Fanuc TP program (LS listing): hs0301h80.ls

/PROG  hs0301h80
/ATTR
COMMENT	= "19-03-01 10:31:46";
PROG_SIZE	= 0;
DEFAULT_GROUP	= 1, 1, *, *, *;
/APPL
    ARC Welding Equipment: 1, *, *, *, *;
/MN
   1:  CALL HOME_ALL;
   1:  UFRAME_NUM = 1;
   1:  UTOOL_NUM = 3;
   1:  COL GUARD ADJUST 150;
   1:  PR[91] = PR[90];
   1:  PR[GP1:91,1] = PR[GP1:90,1] + -1.621;
   1:  PR[GP1:91,2] = PR[GP1:90,2] + 0.568;
   1:  PR[GP1:91,3] = PR[GP1:90,3] + 0.915;
   1:  PR[92] = PR[91];
   1:  PR[GP1:92,3] = PR[GP1:92,3] + 50;
   1:J PR[92] 10% FINE;
   1:L PR[91] R[100]mm/sec CNT100;
   1:  CALL LASER_DRAHT_START;
   1:  PR[GP1:91,1] = PR[GP1:90,1] + -2.739;
   1:  PR[GP1:91,2] = PR[GP1:90,2] + 0.824;
   1:L PR[91] R[100]mm/sec CNT100;
   1:  PR[GP1:91,1] = PR[GP1:90,1] + -3.104;
   1:  PR[GP1:91,2] = PR[GP1:90,2] + 1.033;
   1:L PR[91] R[100]mm/sec CNT100;
   1:  PR[GP1:91,1] = PR[GP1:90,1] + -3.825;
   1:  PR[GP1:91,2] = PR[GP1:90,2] + 1.631;
   1:L PR[91] R[100]mm/sec CNT100;
   1:  PR[GP1:91,1] = PR[GP1:90,1] + -4.095;
   1:  PR[GP1:91,2] = PR[GP1:90,2] + 1.948;
   1:L PR[91] R[100]mm/sec CNT100;
   1:  PR[GP1:91,1] = PR[GP1:90,1] + -4.477;
   1:  PR[GP1:91,2] = PR[GP1:90,2] + 2.812;
   1:L PR[91] R[100]mm/sec CNT100;
   1:  PR[GP1:91,1] = PR[GP1:90,1] + -6.542;
   1:  PR[GP1:91,2] = PR[GP1:90,2] + 8.483;
   1:L PR[91] R[100]mm/sec CNT100;
   1:  PR[GP1:91,1] = PR[GP1:90,1] + -6.656;
   1:  PR[GP1:91,2] = PR[GP1:90,2] + 8.860;
   1:L PR[91] R[100]mm/sec CNT100;
   1:  PR[GP1:91,1] = PR[GP1:90,1] + -6.677;
   1:  PR[GP1:91,2] = PR[GP1:90,2] + 8.904;
   1:L PR[91] R[100]mm/sec CNT100;
   1:  PR[GP1:91,1] = PR[GP1:90,1] + -10.354;
   1:  PR[GP1:91,2] = PR[GP1:90,2] + 13.473;
   1:L PR[91] R[100]mm/sec CNT100;
   1:  PR[GP1:91,1] = PR[GP1:90,1] + -10.502;
   1:  PR[GP1:91,2] = PR[GP1:90,2] + 13.689;
   1:L PR[91] R[100]mm/sec CNT100;
   1:  PR[GP1:91,1] = PR[GP1:90,1] + -10.528;
   1:  PR[GP1:91,2] = PR[GP1:90,2] + 13.715;
   1:L PR[91] R[100]mm/sec CNT100;
   1:  PR[GP1:91,1] = PR[GP1:90,1] + -15.483;
   1:  PR[GP1:91,2] = PR[GP1:90,2] + 16.854;
   1:L PR[91] R[100]mm/sec CNT100;
   1:  PR[GP1:91,1] = PR[GP1:90,1] + -15.694;
   1:  PR[GP1:91,2] = PR[GP1:90,2] + 17.011;
   1:L PR[91] R[100]mm/sec CNT100;
   1:  PR[GP1:91,1] = PR[GP1:90,1] + -15.726;
   1:  PR[GP1:91,2] = PR[GP1:90,2] + 17.028;
   1:L PR[91] R[100]mm/sec CNT100;
   1:  PR[GP1:91,1] = PR[GP1:90,1] + -21.429;
   1:  PR[GP1:91,2] = PR[GP1:90,2] + 18.400;
   1:L PR[91] R[100]mm/sec CNT100;
   1:  PR[GP1:91,1] = PR[GP1:90,1] + -21.680;
   1:  PR[GP1:91,2] = PR[GP1:90,2] + 18.481;
   1:L PR[91] R[100]mm/sec CNT100;
   1:  PR[GP1:91,1] = PR[GP1:90,1] + -21.714;
   1:  PR[GP1:91,2] = PR[GP1:90,2] + 18.486;
   1:L PR[91] R[100]mm/sec CNT100;
   1:  PR[GP1:91,1] = PR[GP1:90,1] + -27.555;
   1:  PR[GP1:91,2] = PR[GP1:90,2] + 17.945;
   1:L PR[91] R[100]mm/sec CNT100;
   1:  PR[GP1:91,1] = PR[GP1:90,1] + -27.820;
   1:  PR[GP1:91,2] = PR[GP1:90,2] + 17.941;
   1:L PR[91] R[100]mm/sec CNT100;
   1:  PR[GP1:91,1] = PR[GP1:90,1] + -27.854;
   1:  PR[GP1:91,2] = PR[GP1:90,2] + 17.935;
   1:L PR[91] R[100]mm/sec CNT100;
   1:  PR[GP1:91,1] = PR[GP1:90,1] + -33.208;
   1:  PR[GP1:91,2] = PR[GP1:90,2] + 15.538;
   1:L PR[91] R[100]mm/sec CNT100;
   1:  PR[GP1:91,1] = PR[GP1:90,1] + -33.458;
   1:  PR[GP1:91,2] = PR[GP1:90,2] + 15.449;
   1:L PR[91] R[100]mm/sec CNT100;
   1:  PR[GP1:91,1] = PR[GP1:90,1] + -33.487;
   1:  PR[GP1:91,2] = PR[GP1:90,2] + 15.433;
   1:L PR[91] R[100]mm/sec CNT100;
   1:  PR[GP1:91,1] = PR[GP1:90,1] + -37.782;
   1:  PR[GP1:91,2] = PR[GP1:90,2] + 11.437;
   1:L PR[91] R[100]mm/sec CNT100;
   1:  PR[GP1:91,1] = PR[GP1:90,1] + -37.990;
   1:  PR[GP1:91,2] = PR[GP1:90,2] + 11.272;
   1:L PR[91] R[100]mm/sec CNT100;
   1:  PR[GP1:91,1] = PR[GP1:90,1] + -38.012;
   1:  PR[GP1:91,2] = PR[GP1:90,2] + 11.247;
   1:L PR[91] R[100]mm/sec CNT100;
   1:  PR[GP1:91,1] = PR[GP1:90,1] + -40.788;
   1:  PR[GP1:91,2] = PR[GP1:90,2] + 6.079;
   1:L PR[91] R[100]mm/sec CNT100;
   1:  PR[GP1:91,1] = PR[GP1:90,1] + -40.932;
   1:  PR[GP1:91,2] = PR[GP1:90,2] + 5.855;
   1:L PR[91] R[100]mm/sec CNT100;
   1:  PR[GP1:91,1] = PR[GP1:90,1] + -40.945;
   1:  PR[GP1:91,2] = PR[GP1:90,2] + 5.826;
   1:L PR[91] R[100]mm/sec CNT100;
   1:  PR[GP1:91,1] = PR[GP1:90,1] + -41.904;
   1:  PR[GP1:91,2] = PR[GP1:90,2] + 0.038;
   1:L PR[91] R[100]mm/sec CNT100;
   1:  PR[GP1:91,1] = PR[GP1:90,1] + -41.969;
   1:  PR[GP1:91,2] = PR[GP1:90,2] + -0.221;
   1:L PR[91] R[100]mm/sec CNT100;
   1:  PR[GP1:91,1] = PR[GP1:90,1] + -41.972;
   1:  PR[GP1:91,2] = PR[GP1:90,2] + -0.252;
   1:L PR[91] R[100]mm/sec CNT100;
   1:  PR[GP1:91,1] = PR[GP1:90,1] + -41.012;
   1:  PR[GP1:91,2] = PR[GP1:90,2] + -6.039;
   1:L PR[91] R[100]mm/sec CNT100;
   1:  PR[GP1:91,1] = PR[GP1:90,1] + -40.991;
   1:  PR[GP1:91,2] = PR[GP1:90,2] + -6.307;
   1:L PR[91] R[100]mm/sec CNT100;
   1:  PR[GP1:91,1] = PR[GP1:90,1] + -40.968;
   1:  PR[GP1:91,2] = PR[GP1:90,2] + -6.395;
   1:L PR[91] R[100]mm/sec CNT100;
   1:  PR[GP1:91,1] = PR[GP1:90,1] + -40.909;
   1:  PR[GP1:91,2] = PR[GP1:90,2] + -6.532;
   1:L PR[91] R[100]mm/sec CNT100;
   1:  PR[GP1:91,1] = PR[GP1:90,1] + -38.133;
   1:  PR[GP1:91,2] = PR[GP1:90,2] + -11.701;
   1:L PR[91] R[100]mm/sec CNT100;
   1:  PR[GP1:91,1] = PR[GP1:90,1] + -38.051;
   1:  PR[GP1:91,2] = PR[GP1:90,2] + -11.828;
   1:L PR[91] R[100]mm/sec CNT100;
   1:  PR[GP1:91,1] = PR[GP1:90,1] + -37.952;
   1:  PR[GP1:91,2] = PR[GP1:90,2] + -11.938;
   1:L PR[91] R[100]mm/sec CNT100;
   1:  PR[GP1:91,1] = PR[GP1:90,1] + -33.656;
   1:  PR[GP1:91,2] = PR[GP1:90,2] + -15.934;
   1:L PR[91] R[100]mm/sec CNT100;
   1:  PR[GP1:91,1] = PR[GP1:90,1] + -33.537;
   1:  PR[GP1:91,2] = PR[GP1:90,2] + -16.029;
   1:L PR[91] R[100]mm/sec CNT100;
   1:  PR[GP1:91,1] = PR[GP1:90,1] + -33.408;
   1:  PR[GP1:91,2] = PR[GP1:90,2] + -16.100;
   1:L PR[91] R[100]mm/sec CNT100;
   1:  PR[GP1:91,1] = PR[GP1:90,1] + -28.053;
   1:  PR[GP1:91,2] = PR[GP1:90,2] + -18.497;
   1:L PR[91] R[100]mm/sec CNT100;
   1:  PR[GP1:91,1] = PR[GP1:90,1] + -27.909;
   1:  PR[GP1:91,2] = PR[GP1:90,2] + -18.549;
   1:L PR[91] R[100]mm/sec CNT100;
   1:  PR[GP1:91,1] = PR[GP1:90,1] + -27.765;
   1:  PR[GP1:91,2] = PR[GP1:90,2] + -18.575;
   1:L PR[91] R[100]mm/sec CNT100;
   1:  PR[GP1:91,1] = PR[GP1:90,1] + -21.923;
   1:  PR[GP1:91,2] = PR[GP1:90,2] + -19.116;
   1:L PR[91] R[100]mm/sec CNT100;
   1:  PR[GP1:91,1] = PR[GP1:90,1] + -21.770;
   1:  PR[GP1:91,2] = PR[GP1:90,2] + -19.118;
   1:L PR[91] R[100]mm/sec CNT100;
   1:  PR[GP1:91,1] = PR[GP1:90,1] + -21.626;
   1:  PR[GP1:91,2] = PR[GP1:90,2] + -19.097;
   1:L PR[91] R[100]mm/sec CNT100;
   1:  PR[GP1:91,1] = PR[GP1:90,1] + -15.922;
   1:  PR[GP1:91,2] = PR[GP1:90,2] + -17.724;
   1:L PR[91] R[100]mm/sec CNT100;
   1:  PR[GP1:91,1] = PR[GP1:90,1] + -15.775;
   1:  PR[GP1:91,2] = PR[GP1:90,2] + -17.677;
   1:L PR[91] R[100]mm/sec CNT100;
   1:  PR[GP1:91,1] = PR[GP1:90,1] + -15.646;
   1:  PR[GP1:91,2] = PR[GP1:90,2] + -17.610;
   1:L PR[91] R[100]mm/sec CNT100;
   1:  PR[GP1:91,1] = PR[GP1:90,1] + -10.691;
   1:  PR[GP1:91,2] = PR[GP1:90,2] + -14.471;
   1:L PR[91] R[100]mm/sec CNT100;
   1:  PR[GP1:91,1] = PR[GP1:90,1] + -10.566;
   1:  PR[GP1:91,2] = PR[GP1:90,2] + -14.378;
   1:L PR[91] R[100]mm/sec CNT100;
   1:  PR[GP1:91,1] = PR[GP1:90,1] + -10.466;
   1:  PR[GP1:91,2] = PR[GP1:90,2] + -14.275;
   1:L PR[91] R[100]mm/sec CNT100;
   1:  PR[GP1:91,1] = PR[GP1:90,1] + -6.788;
   1:  PR[GP1:91,2] = PR[GP1:90,2] + -9.705;
   1:L PR[91] R[100]mm/sec CNT100;
   1:  PR[GP1:91,1] = PR[GP1:90,1] + -6.699;
   1:  PR[GP1:91,2] = PR[GP1:90,2] + -9.576;
   1:L PR[91] R[100]mm/sec CNT100;
   1:  PR[GP1:91,1] = PR[GP1:90,1] + -6.638;
   1:  PR[GP1:91,2] = PR[GP1:90,2] + -9.447;
   1:L PR[91] R[100]mm/sec CNT100;
   1:  PR[GP1:91,1] = PR[GP1:90,1] + -4.634;
   1:  PR[GP1:91,2] = PR[GP1:90,2] + -3.945;
   1:L PR[91] R[100]mm/sec CNT100;
   1:  PR[GP1:91,1] = PR[GP1:90,1] + -4.529;
   1:  PR[GP1:91,2] = PR[GP1:90,2] + -3.569;
   1:L PR[91] R[100]mm/sec CNT100;
   1:  PR[GP1:91,1] = PR[GP1:90,1] + -4.098;
   1:  PR[GP1:91,2] = PR[GP1:90,2] + -2.576;
   1:L PR[91] R[100]mm/sec CNT100;
   1:  PR[GP1:91,1] = PR[GP1:90,1] + -3.825;
   1:  PR[GP1:91,2] = PR[GP1:90,2] + -2.255;
   1:L PR[91] R[100]mm/sec CNT100;
   1:  PR[GP1:91,1] = PR[GP1:90,1] + -3.104;
   1:  PR[GP1:91,2] = PR[GP1:90,2] + -1.657;
   1:L PR[91] R[100]mm/sec CNT100;
   1:  PR[GP1:91,1] = PR[GP1:90,1] + -2.739;
   1:  PR[GP1:91,2] = PR[GP1:90,2] + -1.448;
   1:L PR[91] R[100]mm/sec CNT100;
   1:  PR[GP1:91,1] = PR[GP1:90,1] + -1.621;
   1:  PR[GP1:91,2] = PR[GP1:90,2] + -1.192;
   1:L PR[91] R[100]mm/sec CNT100;
   1:  PR[GP1:91,1] = PR[GP1:90,1] + 1.778;
   1:L PR[91] R[100]mm/sec CNT100;
   1:  PR[GP1:91,1] = PR[GP1:90,1] + 2.895;
   1:  PR[GP1:91,2] = PR[GP1:90,2] + -1.448;
   1:L PR[91] R[100]mm/sec CNT100;
   1:  PR[GP1:91,1] = PR[GP1:90,1] + 3.261;
   1:  PR[GP1:91,2] = PR[GP1:90,2] + -1.657;
   1:L PR[91] R[100]mm/sec CNT100;
   1:  PR[GP1:91,1] = PR[GP1:90,1] + 3.982;
   1:  PR[GP1:91,2] = PR[GP1:90,2] + -2.255;
   1:L PR[91] R[100]mm/sec CNT100;
   1:  PR[GP1:91,1] = PR[GP1:90,1] + 4.252;
   1:  PR[GP1:91,2] = PR[GP1:90,2] + -2.572;
   1:L PR[91] R[100]mm/sec CNT100;
   1:  PR[GP1:91,1] = PR[GP1:90,1] + 4.634;
   1:  PR[GP1:91,2] = PR[GP1:90,2] + -3.436;
   1:L PR[91] R[100]mm/sec CNT100;
   1:  PR[GP1:91,1] = PR[GP1:90,1] + 6.699;
   1:  PR[GP1:91,2] = PR[GP1:90,2] + -9.107;
   1:L PR[91] R[100]mm/sec CNT100;
   1:  PR[GP1:91,1] = PR[GP1:90,1] + 6.813;
   1:  PR[GP1:91,2] = PR[GP1:90,2] + -9.484;
   1:L PR[91] R[100]mm/sec CNT100;
   1:  PR[GP1:91,1] = PR[GP1:90,1] + 6.834;
   1:  PR[GP1:91,2] = PR[GP1:90,2] + -9.528;
   1:L PR[91] R[100]mm/sec CNT100;
   1:  PR[GP1:91,1] = PR[GP1:90,1] + 10.510;
   1:  PR[GP1:91,2] = PR[GP1:90,2] + -14.097;
   1:L PR[91] R[100]mm/sec CNT100;
   1:  PR[GP1:91,1] = PR[GP1:90,1] + 10.659;
   1:  PR[GP1:91,2] = PR[GP1:90,2] + -14.313;
   1:L PR[91] R[100]mm/sec CNT100;
   1:  PR[GP1:91,1] = PR[GP1:90,1] + 10.685;
   1:  PR[GP1:91,2] = PR[GP1:90,2] + -14.339;
   1:L PR[91] R[100]mm/sec CNT100;
   1:  PR[GP1:91,1] = PR[GP1:90,1] + 15.640;
   1:  PR[GP1:91,2] = PR[GP1:90,2] + -17.478;
   1:L PR[91] R[100]mm/sec CNT100;
   1:  PR[GP1:91,1] = PR[GP1:90,1] + 15.851;
   1:  PR[GP1:91,2] = PR[GP1:90,2] + -17.635;
   1:L PR[91] R[100]mm/sec CNT100;
   1:  PR[GP1:91,1] = PR[GP1:90,1] + 15.883;
   1:  PR[GP1:91,2] = PR[GP1:90,2] + -17.652;
   1:L PR[91] R[100]mm/sec CNT100;
   1:  PR[GP1:91,1] = PR[GP1:90,1] + 21.586;
   1:  PR[GP1:91,2] = PR[GP1:90,2] + -19.024;
   1:L PR[91] R[100]mm/sec CNT100;
   1:  PR[GP1:91,1] = PR[GP1:90,1] + 21.836;
   1:  PR[GP1:91,2] = PR[GP1:90,2] + -19.105;
   1:L PR[91] R[100]mm/sec CNT100;
   1:  PR[GP1:91,1] = PR[GP1:90,1] + 21.871;
   1:  PR[GP1:91,2] = PR[GP1:90,2] + -19.110;
   1:L PR[91] R[100]mm/sec CNT100;
   1:  PR[GP1:91,1] = PR[GP1:90,1] + 27.712;
   1:  PR[GP1:91,2] = PR[GP1:90,2] + -18.569;
   1:L PR[91] R[100]mm/sec CNT100;
   1:  PR[GP1:91,1] = PR[GP1:90,1] + 27.976;
   1:  PR[GP1:91,2] = PR[GP1:90,2] + -18.565;
   1:L PR[91] R[100]mm/sec CNT100;
   1:  PR[GP1:91,1] = PR[GP1:90,1] + 28.010;
   1:  PR[GP1:91,2] = PR[GP1:90,2] + -18.559;
   1:L PR[91] R[100]mm/sec CNT100;
   1:  PR[GP1:91,1] = PR[GP1:90,1] + 33.365;
   1:  PR[GP1:91,2] = PR[GP1:90,2] + -16.162;
   1:L PR[91] R[100]mm/sec CNT100;
   1:  PR[GP1:91,1] = PR[GP1:90,1] + 33.614;
   1:  PR[GP1:91,2] = PR[GP1:90,2] + -16.073;
   1:L PR[91] R[100]mm/sec CNT100;
   1:  PR[GP1:91,1] = PR[GP1:90,1] + 33.644;
   1:  PR[GP1:91,2] = PR[GP1:90,2] + -16.057;
   1:L PR[91] R[100]mm/sec CNT100;
   1:  PR[GP1:91,1] = PR[GP1:90,1] + 37.938;
   1:  PR[GP1:91,2] = PR[GP1:90,2] + -12.061;
   1:L PR[91] R[100]mm/sec CNT100;
   1:  PR[GP1:91,1] = PR[GP1:90,1] + 38.147;
   1:  PR[GP1:91,2] = PR[GP1:90,2] + -11.895;
   1:L PR[91] R[100]mm/sec CNT100;
   1:  PR[GP1:91,1] = PR[GP1:90,1] + 38.169;
   1:  PR[GP1:91,2] = PR[GP1:90,2] + -11.871;
   1:L PR[91] R[100]mm/sec CNT100;
   1:  PR[GP1:91,1] = PR[GP1:90,1] + 40.944;
   1:  PR[GP1:91,2] = PR[GP1:90,2] + -6.703;
   1:L PR[91] R[100]mm/sec CNT100;
   1:  PR[GP1:91,1] = PR[GP1:90,1] + 41.089;
   1:  PR[GP1:91,2] = PR[GP1:90,2] + -6.479;
   1:L PR[91] R[100]mm/sec CNT100;
   1:  PR[GP1:91,1] = PR[GP1:90,1] + 41.102;
   1:  PR[GP1:91,2] = PR[GP1:90,2] + -6.450;
   1:L PR[91] R[100]mm/sec CNT100;
   1:  PR[GP1:91,1] = PR[GP1:90,1] + 42.061;
   1:  PR[GP1:91,2] = PR[GP1:90,2] + -0.662;
   1:L PR[91] R[100]mm/sec CNT100;
   1:  PR[GP1:91,1] = PR[GP1:90,1] + 42.126;
   1:  PR[GP1:91,2] = PR[GP1:90,2] + -0.403;
   1:L PR[91] R[100]mm/sec CNT100;
   1:  PR[GP1:91,1] = PR[GP1:90,1] + 42.129;
   1:  PR[GP1:91,2] = PR[GP1:90,2] + -0.372;
   1:L PR[91] R[100]mm/sec CNT100;
   1:  PR[GP1:91,1] = PR[GP1:90,1] + 41.169;
   1:  PR[GP1:91,2] = PR[GP1:90,2] + 5.415;
   1:L PR[91] R[100]mm/sec CNT100;
   1:  PR[GP1:91,1] = PR[GP1:90,1] + 41.147;
   1:  PR[GP1:91,2] = PR[GP1:90,2] + 5.683;
   1:L PR[91] R[100]mm/sec CNT100;
   1:  PR[GP1:91,1] = PR[GP1:90,1] + 41.125;
   1:  PR[GP1:91,2] = PR[GP1:90,2] + 5.771;
   1:L PR[91] R[100]mm/sec CNT100;
   1:  PR[GP1:91,1] = PR[GP1:90,1] + 41.066;
   1:  PR[GP1:91,2] = PR[GP1:90,2] + 5.908;
   1:L PR[91] R[100]mm/sec CNT100;
   1:  PR[GP1:91,1] = PR[GP1:90,1] + 38.290;
   1:  PR[GP1:91,2] = PR[GP1:90,2] + 11.077;
   1:L PR[91] R[100]mm/sec CNT100;
   1:  PR[GP1:91,1] = PR[GP1:90,1] + 38.208;
   1:  PR[GP1:91,2] = PR[GP1:90,2] + 11.204;
   1:L PR[91] R[100]mm/sec CNT100;
   1:  PR[GP1:91,1] = PR[GP1:90,1] + 38.108;
   1:  PR[GP1:91,2] = PR[GP1:90,2] + 11.314;
   1:L PR[91] R[100]mm/sec CNT100;
   1:  PR[GP1:91,1] = PR[GP1:90,1] + 33.813;
   1:  PR[GP1:91,2] = PR[GP1:90,2] + 15.310;
   1:L PR[91] R[100]mm/sec CNT100;
   1:  PR[GP1:91,1] = PR[GP1:90,1] + 33.694;
   1:  PR[GP1:91,2] = PR[GP1:90,2] + 15.405;
   1:L PR[91] R[100]mm/sec CNT100;
   1:  PR[GP1:91,1] = PR[GP1:90,1] + 33.565;
   1:  PR[GP1:91,2] = PR[GP1:90,2] + 15.476;
   1:L PR[91] R[100]mm/sec CNT100;
   1:  PR[GP1:91,1] = PR[GP1:90,1] + 28.210;
   1:  PR[GP1:91,2] = PR[GP1:90,2] + 17.873;
   1:L PR[91] R[100]mm/sec CNT100;
   1:  PR[GP1:91,1] = PR[GP1:90,1] + 28.066;
   1:  PR[GP1:91,2] = PR[GP1:90,2] + 17.925;
   1:L PR[91] R[100]mm/sec CNT100;
   1:  PR[GP1:91,1] = PR[GP1:90,1] + 27.922;
   1:  PR[GP1:91,2] = PR[GP1:90,2] + 17.951;
   1:L PR[91] R[100]mm/sec CNT100;
   1:  PR[GP1:91,1] = PR[GP1:90,1] + 22.080;
   1:  PR[GP1:91,2] = PR[GP1:90,2] + 18.492;
   1:L PR[91] R[100]mm/sec CNT100;
   1:  PR[GP1:91,1] = PR[GP1:90,1] + 21.926;
   1:  PR[GP1:91,2] = PR[GP1:90,2] + 18.494;
   1:L PR[91] R[100]mm/sec CNT100;
   1:  PR[GP1:91,1] = PR[GP1:90,1] + 21.782;
   1:  PR[GP1:91,2] = PR[GP1:90,2] + 18.473;
   1:L PR[91] R[100]mm/sec CNT100;
   1:  PR[GP1:91,1] = PR[GP1:90,1] + 16.079;
   1:  PR[GP1:91,2] = PR[GP1:90,2] + 17.100;
   1:L PR[91] R[100]mm/sec CNT100;
   1:  PR[GP1:91,1] = PR[GP1:90,1] + 15.931;
   1:  PR[GP1:91,2] = PR[GP1:90,2] + 17.053;
   1:L PR[91] R[100]mm/sec CNT100;
   1:  PR[GP1:91,1] = PR[GP1:90,1] + 15.803;
   1:  PR[GP1:91,2] = PR[GP1:90,2] + 16.986;
   1:L PR[91] R[100]mm/sec CNT100;
   1:  PR[GP1:91,1] = PR[GP1:90,1] + 10.847;
   1:  PR[GP1:91,2] = PR[GP1:90,2] + 13.847;
   1:L PR[91] R[100]mm/sec CNT100;
   1:  PR[GP1:91,1] = PR[GP1:90,1] + 10.722;
   1:  PR[GP1:91,2] = PR[GP1:90,2] + 13.754;
   1:L PR[91] R[100]mm/sec CNT100;
   1:  PR[GP1:91,1] = PR[GP1:90,1] + 10.622;
   1:  PR[GP1:91,2] = PR[GP1:90,2] + 13.651;
   1:L PR[91] R[100]mm/sec CNT100;
   1:  PR[GP1:91,1] = PR[GP1:90,1] + 6.945;
   1:  PR[GP1:91,2] = PR[GP1:90,2] + 9.081;
   1:L PR[91] R[100]mm/sec CNT100;
   1:  PR[GP1:91,1] = PR[GP1:90,1] + 6.856;
   1:  PR[GP1:91,2] = PR[GP1:90,2] + 8.952;
   1:L PR[91] R[100]mm/sec CNT100;
   1:  PR[GP1:91,1] = PR[GP1:90,1] + 6.795;
   1:  PR[GP1:91,2] = PR[GP1:90,2] + 8.823;
   1:L PR[91] R[100]mm/sec CNT100;
   1:  PR[GP1:91,1] = PR[GP1:90,1] + 4.791;
   1:  PR[GP1:91,2] = PR[GP1:90,2] + 3.321;
   1:L PR[91] R[100]mm/sec CNT100;
   1:  PR[GP1:91,1] = PR[GP1:90,1] + 4.686;
   1:  PR[GP1:91,2] = PR[GP1:90,2] + 2.945;
   1:L PR[91] R[100]mm/sec CNT100;
   1:  PR[GP1:91,1] = PR[GP1:90,1] + 4.255;
   1:  PR[GP1:91,2] = PR[GP1:90,2] + 1.952;
   1:L PR[91] R[100]mm/sec CNT100;
   1:  PR[GP1:91,1] = PR[GP1:90,1] + 3.982;
   1:  PR[GP1:91,2] = PR[GP1:90,2] + 1.631;
   1:L PR[91] R[100]mm/sec CNT100;
   1:  PR[GP1:91,1] = PR[GP1:90,1] + 3.261;
   1:  PR[GP1:91,2] = PR[GP1:90,2] + 1.033;
   1:L PR[91] R[100]mm/sec CNT100;
   1:  PR[GP1:91,1] = PR[GP1:90,1] + 2.895;
   1:  PR[GP1:91,2] = PR[GP1:90,2] + 0.824;
   1:L PR[91] R[100]mm/sec CNT100;
   1:  PR[GP1:91,1] = PR[GP1:90,1] + 1.778;
   1:  PR[GP1:91,2] = PR[GP1:90,2] + 0.568;
   1:L PR[91] R[100]mm/sec CNT100;
   1:  PR[GP1:91,1] = PR[GP1:90,1] + -1.621;
   1:L PR[91] R[100]mm/sec CNT100;
   1:  PR[91] = PR[90];
   1:  PR[GP1:91,1] = PR[GP1:90,1] + -2.689;
   1:  PR[GP1:91,2] = PR[GP1:90,2] + 0.801;
   1:  PR[GP1:91,3] = PR[GP1:90,3] + 1.525;
   1:L PR[91] R[100]mm/sec CNT100;
   1:  PR[GP1:91,1] = PR[GP1:90,1] + -3.181;
   1:  PR[GP1:91,2] = PR[GP1:90,2] + 1.083;
   1:L PR[91] R[100]mm/sec CNT100;
   1:  PR[GP1:91,1] = PR[GP1:90,1] + -3.762;
   1:  PR[GP1:91,2] = PR[GP1:90,2] + 1.565;
   1:L PR[91] R[100]mm/sec CNT100;
   1:  PR[GP1:91,1] = PR[GP1:90,1] + -4.129;
   1:  PR[GP1:91,2] = PR[GP1:90,2] + 1.996;
   1:L PR[91] R[100]mm/sec CNT100;
   1:  PR[GP1:91,1] = PR[GP1:90,1] + -4.510;
   1:  PR[GP1:91,2] = PR[GP1:90,2] + 2.901;
   1:L PR[91] R[100]mm/sec CNT100;
   1:  PR[GP1:91,1] = PR[GP1:90,1] + -5.965;
   1:  PR[GP1:91,2] = PR[GP1:90,2] + 6.895;
   1:L PR[91] R[100]mm/sec CNT100;
   1:  PR[GP1:91,1] = PR[GP1:90,1] + -6.225;
   1:  PR[GP1:91,2] = PR[GP1:90,2] + 7.635;
   1:L PR[91] R[100]mm/sec CNT100;
   1:  PR[GP1:91,1] = PR[GP1:90,1] + -6.443;
   1:  PR[GP1:91,2] = PR[GP1:90,2] + 8.403;
   1:L PR[91] R[100]mm/sec CNT100;
   1:  PR[GP1:91,1] = PR[GP1:90,1] + -6.692;
   1:  PR[GP1:91,2] = PR[GP1:90,2] + 8.931;
   1:L PR[91] R[100]mm/sec CNT100;
   1:  PR[GP1:91,1] = PR[GP1:90,1] + -9.685;
   1:  PR[GP1:91,2] = PR[GP1:90,2] + 12.650;
   1:L PR[91] R[100]mm/sec CNT100;
   1:  PR[GP1:91,1] = PR[GP1:90,1] + -10.144;
   1:  PR[GP1:91,2] = PR[GP1:90,2] + 13.314;
   1:L PR[91] R[100]mm/sec CNT100;
   1:  PR[GP1:91,1] = PR[GP1:90,1] + -10.548;
   1:  PR[GP1:91,2] = PR[GP1:90,2] + 13.733;
   1:L PR[91] R[100]mm/sec CNT100;
   1:  PR[GP1:91,1] = PR[GP1:90,1] + -14.582;
   1:  PR[GP1:91,2] = PR[GP1:90,2] + 16.288;
   1:L PR[91] R[100]mm/sec CNT100;
   1:  PR[GP1:91,1] = PR[GP1:90,1] + -15.230;
   1:  PR[GP1:91,2] = PR[GP1:90,2] + 16.770;
   1:L PR[91] R[100]mm/sec CNT100;
   1:  PR[GP1:91,1] = PR[GP1:90,1] + -15.747;
   1:  PR[GP1:91,2] = PR[GP1:90,2] + 17.037;
   1:L PR[91] R[100]mm/sec CNT100;
   1:  PR[GP1:91,1] = PR[GP1:90,1] + -20.390;
   1:  PR[GP1:91,2] = PR[GP1:90,2] + 18.154;
   1:L PR[91] R[100]mm/sec CNT100;
   1:  PR[GP1:91,1] = PR[GP1:90,1] + -21.159;
   1:  PR[GP1:91,2] = PR[GP1:90,2] + 18.402;
   1:L PR[91] R[100]mm/sec CNT100;
   1:  PR[GP1:91,1] = PR[GP1:90,1] + -21.734;
   1:  PR[GP1:91,2] = PR[GP1:90,2] + 18.488;
   1:L PR[91] R[100]mm/sec CNT100;
   1:  PR[GP1:91,1] = PR[GP1:90,1] + -26.488;
   1:  PR[GP1:91,2] = PR[GP1:90,2] + 18.047;
   1:L PR[91] R[100]mm/sec CNT100;
   1:  PR[GP1:91,1] = PR[GP1:90,1] + -27.298;
   1:  PR[GP1:91,2] = PR[GP1:90,2] + 18.035;
   1:L PR[91] R[100]mm/sec CNT100;
   1:  PR[GP1:91,1] = PR[GP1:90,1] + -27.869;
   1:  PR[GP1:91,2] = PR[GP1:90,2] + 17.931;
   1:L PR[91] R[100]mm/sec CNT100;
   1:  PR[GP1:91,1] = PR[GP1:90,1] + -32.227;
   1:  PR[GP1:91,2] = PR[GP1:90,2] + 15.980;
   1:L PR[91] R[100]mm/sec CNT100;
   1:  PR[GP1:91,1] = PR[GP1:90,1] + -32.990;
   1:  PR[GP1:91,2] = PR[GP1:90,2] + 15.708;
   1:L PR[91] R[100]mm/sec CNT100;
   1:  PR[GP1:91,1] = PR[GP1:90,1] + -33.497;
   1:  PR[GP1:91,2] = PR[GP1:90,2] + 15.426;
   1:L PR[91] R[100]mm/sec CNT100;
   1:  PR[GP1:91,1] = PR[GP1:90,1] + -36.993;
   1:  PR[GP1:91,2] = PR[GP1:90,2] + 12.174;
   1:L PR[91] R[100]mm/sec CNT100;
   1:  PR[GP1:91,1] = PR[GP1:90,1] + -37.628;
   1:  PR[GP1:91,2] = PR[GP1:90,2] + 11.669;
   1:L PR[91] R[100]mm/sec CNT100;
   1:  PR[GP1:91,1] = PR[GP1:90,1] + -38.017;
   1:  PR[GP1:91,2] = PR[GP1:90,2] + 11.241;
   1:L PR[91] R[100]mm/sec CNT100;
   1:  PR[GP1:91,1] = PR[GP1:90,1] + -40.276;
   1:  PR[GP1:91,2] = PR[GP1:90,2] + 7.034;
   1:L PR[91] R[100]mm/sec CNT100;
   1:  PR[GP1:91,1] = PR[GP1:90,1] + -40.716;
   1:  PR[GP1:91,2] = PR[GP1:90,2] + 6.352;
   1:L PR[91] R[100]mm/sec CNT100;
   1:  PR[GP1:91,1] = PR[GP1:90,1] + -40.946;
   1:  PR[GP1:91,2] = PR[GP1:90,2] + 5.822;
   1:L PR[91] R[100]mm/sec CNT100;
   1:  PR[GP1:91,1] = PR[GP1:90,1] + -41.727;
   1:  PR[GP1:91,2] = PR[GP1:90,2] + 1.111;
   1:L PR[91] R[100]mm/sec CNT100;
   1:  PR[GP1:91,1] = PR[GP1:90,1] + -41.925;
   1:  PR[GP1:91,2] = PR[GP1:90,2] + 0.322;
   1:L PR[91] R[100]mm/sec CNT100;
   1:  PR[GP1:91,1] = PR[GP1:90,1] + -41.972;
   1:  PR[GP1:91,2] = PR[GP1:90,2] + -0.252;
   1:L PR[91] R[100]mm/sec CNT100;
   1:  PR[GP1:91,1] = PR[GP1:90,1] + -41.191;
   1:  PR[GP1:91,2] = PR[GP1:90,2] + -4.963;
   1:L PR[91] R[100]mm/sec CNT100;
   1:  PR[GP1:91,1] = PR[GP1:90,1] + -41.124;
   1:  PR[GP1:91,2] = PR[GP1:90,2] + -5.774;
   1:L PR[91] R[100]mm/sec CNT100;
   1:  PR[GP1:91,1] = PR[GP1:90,1] + -40.970;
   1:  PR[GP1:91,2] = PR[GP1:90,2] + -6.392;
   1:L PR[91] R[100]mm/sec CNT100;
   1:  PR[GP1:91,1] = PR[GP1:90,1] + -40.693;
   1:  PR[GP1:91,2] = PR[GP1:90,2] + -7.029;
   1:L PR[91] R[100]mm/sec CNT100;
   1:  PR[GP1:91,1] = PR[GP1:90,1] + -38.434;
   1:  PR[GP1:91,2] = PR[GP1:90,2] + -11.236;
   1:L PR[91] R[100]mm/sec CNT100;
   1:  PR[GP1:91,1] = PR[GP1:90,1] + -38.056;
   1:  PR[GP1:91,2] = PR[GP1:90,2] + -11.822;
   1:L PR[91] R[100]mm/sec CNT100;
   1:  PR[GP1:91,1] = PR[GP1:90,1] + -37.590;
   1:  PR[GP1:91,2] = PR[GP1:90,2] + -12.336;
   1:L PR[91] R[100]mm/sec CNT100;
   1:  PR[GP1:91,1] = PR[GP1:90,1] + -34.094;
   1:  PR[GP1:91,2] = PR[GP1:90,2] + -15.589;
   1:L PR[91] R[100]mm/sec CNT100;
   1:  PR[GP1:91,1] = PR[GP1:90,1] + -33.547;
   1:  PR[GP1:91,2] = PR[GP1:90,2] + -16.023;
   1:L PR[91] R[100]mm/sec CNT100;
   1:  PR[GP1:91,1] = PR[GP1:90,1] + -32.941;
   1:  PR[GP1:91,2] = PR[GP1:90,2] + -16.359;
   1:L PR[91] R[100]mm/sec CNT100;
   1:  PR[GP1:91,1] = PR[GP1:90,1] + -28.582;
   1:  PR[GP1:91,2] = PR[GP1:90,2] + -18.310;
   1:L PR[91] R[100]mm/sec CNT100;
   1:  PR[GP1:91,1] = PR[GP1:90,1] + -27.924;
   1:  PR[GP1:91,2] = PR[GP1:90,2] + -18.545;
   1:L PR[91] R[100]mm/sec CNT100;
   1:  PR[GP1:91,1] = PR[GP1:90,1] + -27.244;
   1:  PR[GP1:91,2] = PR[GP1:90,2] + -18.668;
   1:L PR[91] R[100]mm/sec CNT100;
   1:  PR[GP1:91,1] = PR[GP1:90,1] + -22.488;
   1:  PR[GP1:91,2] = PR[GP1:90,2] + -19.109;
   1:L PR[91] R[100]mm/sec CNT100;
   1:  PR[GP1:91,1] = PR[GP1:90,1] + -21.789;
   1:  PR[GP1:91,2] = PR[GP1:90,2] + -19.120;
   1:L PR[91] R[100]mm/sec CNT100;
   1:  PR[GP1:91,1] = PR[GP1:90,1] + -21.106;
   1:  PR[GP1:91,2] = PR[GP1:90,2] + -19.018;
   1:L PR[91] R[100]mm/sec CNT100;
   1:  PR[GP1:91,1] = PR[GP1:90,1] + -16.463;
   1:  PR[GP1:91,2] = PR[GP1:90,2] + -17.900;
   1:L PR[91] R[100]mm/sec CNT100;
   1:  PR[GP1:91,1] = PR[GP1:90,1] + -15.796;
   1:  PR[GP1:91,2] = PR[GP1:90,2] + -17.686;
   1:L PR[91] R[100]mm/sec CNT100;
   1:  PR[GP1:91,1] = PR[GP1:90,1] + -15.182;
   1:  PR[GP1:91,2] = PR[GP1:90,2] + -17.370;
   1:L PR[91] R[100]mm/sec CNT100;
   1:  PR[GP1:91,1] = PR[GP1:90,1] + -11.149;
   1:  PR[GP1:91,2] = PR[GP1:90,2] + -14.814;
   1:L PR[91] R[100]mm/sec CNT100;
   1:  PR[GP1:91,1] = PR[GP1:90,1] + -10.586;
   1:  PR[GP1:91,2] = PR[GP1:90,2] + -14.396;
   1:L PR[91] R[100]mm/sec CNT100;
   1:  PR[GP1:91,1] = PR[GP1:90,1] + -10.107;
   1:  PR[GP1:91,2] = PR[GP1:90,2] + -13.900;
   1:L PR[91] R[100]mm/sec CNT100;
   1:  PR[GP1:91,1] = PR[GP1:90,1] + -7.114;
   1:  PR[GP1:91,2] = PR[GP1:90,2] + -10.181;
   1:L PR[91] R[100]mm/sec CNT100;
   1:  PR[GP1:91,1] = PR[GP1:90,1] + -6.715;
   1:  PR[GP1:91,2] = PR[GP1:90,2] + -9.603;
   1:L PR[91] R[100]mm/sec CNT100;
   1:  PR[GP1:91,1] = PR[GP1:90,1] + -6.421;
   1:  PR[GP1:91,2] = PR[GP1:90,2] + -8.980;
   1:L PR[91] R[100]mm/sec CNT100;
   1:  PR[GP1:91,1] = PR[GP1:90,1] + -4.790;
   1:  PR[GP1:91,2] = PR[GP1:90,2] + -4.502;
   1:L PR[91] R[100]mm/sec CNT100;
   1:  PR[GP1:91,1] = PR[GP1:90,1] + -4.532;
   1:  PR[GP1:91,2] = PR[GP1:90,2] + -3.577;
   1:L PR[91] R[100]mm/sec CNT100;
   1:  PR[GP1:91,1] = PR[GP1:90,1] + -4.129;
   1:  PR[GP1:91,2] = PR[GP1:90,2] + -2.620;
   1:L PR[91] R[100]mm/sec CNT100;
   1:  PR[GP1:91,1] = PR[GP1:90,1] + -3.762;
   1:  PR[GP1:91,2] = PR[GP1:90,2] + -2.189;
   1:L PR[91] R[100]mm/sec CNT100;
   1:  PR[GP1:91,1] = PR[GP1:90,1] + -3.181;
   1:  PR[GP1:91,2] = PR[GP1:90,2] + -1.707;
   1:L PR[91] R[100]mm/sec CNT100;
   1:  PR[GP1:91,1] = PR[GP1:90,1] + -2.689;
   1:  PR[GP1:91,2] = PR[GP1:90,2] + -1.425;
   1:L PR[91] R[100]mm/sec CNT100;
   1:  PR[GP1:91,1] = PR[GP1:90,1] + -1.613;
   1:  PR[GP1:91,2] = PR[GP1:90,2] + -1.192;
   1:L PR[91] R[100]mm/sec CNT100;
   1:  PR[GP1:91,1] = PR[GP1:90,1] + 1.770;
   1:L PR[91] R[100]mm/sec CNT100;
   1:  PR[GP1:91,1] = PR[GP1:90,1] + 2.846;
   1:  PR[GP1:91,2] = PR[GP1:90,2] + -1.425;
   1:L PR[91] R[100]mm/sec CNT100;
   1:  PR[GP1:91,1] = PR[GP1:90,1] + 3.338;
   1:  PR[GP1:91,2] = PR[GP1:90,2] + -1.707;
   1:L PR[91] R[100]mm/sec CNT100;
   1:  PR[GP1:91,1] = PR[GP1:90,1] + 3.919;
   1:  PR[GP1:91,2] = PR[GP1:90,2] + -2.189;
   1:L PR[91] R[100]mm/sec CNT100;
   1:  PR[GP1:91,1] = PR[GP1:90,1] + 4.285;
   1:  PR[GP1:91,2] = PR[GP1:90,2] + -2.620;
   1:L PR[91] R[100]mm/sec CNT100;
   1:  PR[GP1:91,1] = PR[GP1:90,1] + 4.667;
   1:  PR[GP1:91,2] = PR[GP1:90,2] + -3.525;
   1:L PR[91] R[100]mm/sec CNT100;
   1:  PR[GP1:91,1] = PR[GP1:90,1] + 6.251;
   1:  PR[GP1:91,2] = PR[GP1:90,2] + -7.882;
   1:L PR[91] R[100]mm/sec CNT100;
   1:  PR[GP1:91,1] = PR[GP1:90,1] + 6.383;
   1:  PR[GP1:91,2] = PR[GP1:90,2] + -8.264;
   1:L PR[91] R[100]mm/sec CNT100;
   1:  PR[GP1:91,1] = PR[GP1:90,1] + 6.600;
   1:  PR[GP1:91,2] = PR[GP1:90,2] + -9.027;
   1:L PR[91] R[100]mm/sec CNT100;
   1:  PR[GP1:91,1] = PR[GP1:90,1] + 6.849;
   1:  PR[GP1:91,2] = PR[GP1:90,2] + -9.555;
   1:L PR[91] R[100]mm/sec CNT100;
   1:  PR[GP1:91,1] = PR[GP1:90,1] + 9.842;
   1:  PR[GP1:91,2] = PR[GP1:90,2] + -13.274;
   1:L PR[91] R[100]mm/sec CNT100;
   1:  PR[GP1:91,1] = PR[GP1:90,1] + 10.301;
   1:  PR[GP1:91,2] = PR[GP1:90,2] + -13.938;
   1:L PR[91] R[100]mm/sec CNT100;
   1:  PR[GP1:91,1] = PR[GP1:90,1] + 10.705;
   1:  PR[GP1:91,2] = PR[GP1:90,2] + -14.357;
   1:L PR[91] R[100]mm/sec CNT100;
   1:  PR[GP1:91,1] = PR[GP1:90,1] + 14.738;
   1:  PR[GP1:91,2] = PR[GP1:90,2] + -16.912;
   1:L PR[91] R[100]mm/sec CNT100;
   1:  PR[GP1:91,1] = PR[GP1:90,1] + 15.387;
   1:  PR[GP1:91,2] = PR[GP1:90,2] + -17.394;
   1:L PR[91] R[100]mm/sec CNT100;
   1:  PR[GP1:91,1] = PR[GP1:90,1] + 15.904;
   1:  PR[GP1:91,2] = PR[GP1:90,2] + -17.661;
   1:L PR[91] R[100]mm/sec CNT100;
   1:  PR[GP1:91,1] = PR[GP1:90,1] + 20.546;
   1:  PR[GP1:91,2] = PR[GP1:90,2] + -18.778;
   1:L PR[91] R[100]mm/sec CNT100;
   1:  PR[GP1:91,1] = PR[GP1:90,1] + 21.316;
   1:  PR[GP1:91,2] = PR[GP1:90,2] + -19.026;
   1:L PR[91] R[100]mm/sec CNT100;
   1:  PR[GP1:91,1] = PR[GP1:90,1] + 21.891;
   1:  PR[GP1:91,2] = PR[GP1:90,2] + -19.112;
   1:L PR[91] R[100]mm/sec CNT100;
   1:  PR[GP1:91,1] = PR[GP1:90,1] + 26.645;
   1:  PR[GP1:91,2] = PR[GP1:90,2] + -18.671;
   1:L PR[91] R[100]mm/sec CNT100;
   1:  PR[GP1:91,1] = PR[GP1:90,1] + 27.455;
   1:  PR[GP1:91,2] = PR[GP1:90,2] + -18.659;
   1:L PR[91] R[100]mm/sec CNT100;
   1:  PR[GP1:91,1] = PR[GP1:90,1] + 28.026;
   1:  PR[GP1:91,2] = PR[GP1:90,2] + -18.555;
   1:L PR[91] R[100]mm/sec CNT100;
   1:  PR[GP1:91,1] = PR[GP1:90,1] + 32.384;
   1:  PR[GP1:91,2] = PR[GP1:90,2] + -16.604;
   1:L PR[91] R[100]mm/sec CNT100;
   1:  PR[GP1:91,1] = PR[GP1:90,1] + 33.147;
   1:  PR[GP1:91,2] = PR[GP1:90,2] + -16.331;
   1:L PR[91] R[100]mm/sec CNT100;
   1:  PR[GP1:91,1] = PR[GP1:90,1] + 33.654;
   1:  PR[GP1:91,2] = PR[GP1:90,2] + -16.050;
   1:L PR[91] R[100]mm/sec CNT100;
   1:  PR[GP1:91,1] = PR[GP1:90,1] + 37.149;
   1:  PR[GP1:91,2] = PR[GP1:90,2] + -12.798;
   1:L PR[91] R[100]mm/sec CNT100;
   1:  PR[GP1:91,1] = PR[GP1:90,1] + 37.785;
   1:  PR[GP1:91,2] = PR[GP1:90,2] + -12.293;
   1:L PR[91] R[100]mm/sec CNT100;
   1:  PR[GP1:91,1] = PR[GP1:90,1] + 38.174;
   1:  PR[GP1:91,2] = PR[GP1:90,2] + -11.865;
   1:L PR[91] R[100]mm/sec CNT100;
   1:  PR[GP1:91,1] = PR[GP1:90,1] + 40.433;
   1:  PR[GP1:91,2] = PR[GP1:90,2] + -7.658;
   1:L PR[91] R[100]mm/sec CNT100;
   1:  PR[GP1:91,1] = PR[GP1:90,1] + 40.873;
   1:  PR[GP1:91,2] = PR[GP1:90,2] + -6.976;
   1:L PR[91] R[100]mm/sec CNT100;
   1:  PR[GP1:91,1] = PR[GP1:90,1] + 41.103;
   1:  PR[GP1:91,2] = PR[GP1:90,2] + -6.446;
   1:L PR[91] R[100]mm/sec CNT100;
   1:  PR[GP1:91,1] = PR[GP1:90,1] + 41.884;
   1:  PR[GP1:91,2] = PR[GP1:90,2] + -1.735;
   1:L PR[91] R[100]mm/sec CNT100;
   1:  PR[GP1:91,1] = PR[GP1:90,1] + 42.082;
   1:  PR[GP1:91,2] = PR[GP1:90,2] + -0.946;
   1:L PR[91] R[100]mm/sec CNT100;
   1:  PR[GP1:91,1] = PR[GP1:90,1] + 42.129;
   1:  PR[GP1:91,2] = PR[GP1:90,2] + -0.372;
   1:L PR[91] R[100]mm/sec CNT100;
   1:  PR[GP1:91,1] = PR[GP1:90,1] + 41.348;
   1:  PR[GP1:91,2] = PR[GP1:90,2] + 4.339;
   1:L PR[91] R[100]mm/sec CNT100;
   1:  PR[GP1:91,1] = PR[GP1:90,1] + 41.281;
   1:  PR[GP1:91,2] = PR[GP1:90,2] + 5.150;
   1:L PR[91] R[100]mm/sec CNT100;
   1:  PR[GP1:91,1] = PR[GP1:90,1] + 41.126;
   1:  PR[GP1:91,2] = PR[GP1:90,2] + 5.768;
   1:L PR[91] R[100]mm/sec CNT100;
   1:  PR[GP1:91,1] = PR[GP1:90,1] + 40.850;
   1:  PR[GP1:91,2] = PR[GP1:90,2] + 6.405;
   1:L PR[91] R[100]mm/sec CNT100;
   1:  PR[GP1:91,1] = PR[GP1:90,1] + 38.591;
   1:  PR[GP1:91,2] = PR[GP1:90,2] + 10.612;
   1:L PR[91] R[100]mm/sec CNT100;
   1:  PR[GP1:91,1] = PR[GP1:90,1] + 38.213;
   1:  PR[GP1:91,2] = PR[GP1:90,2] + 11.198;
   1:L PR[91] R[100]mm/sec CNT100;
   1:  PR[GP1:91,1] = PR[GP1:90,1] + 37.747;
   1:  PR[GP1:91,2] = PR[GP1:90,2] + 11.712;
   1:L PR[91] R[100]mm/sec CNT100;
   1:  PR[GP1:91,1] = PR[GP1:90,1] + 34.250;
   1:  PR[GP1:91,2] = PR[GP1:90,2] + 14.965;
   1:L PR[91] R[100]mm/sec CNT100;
   1:  PR[GP1:91,1] = PR[GP1:90,1] + 33.704;
   1:  PR[GP1:91,2] = PR[GP1:90,2] + 15.399;
   1:L PR[91] R[100]mm/sec CNT100;
   1:  PR[GP1:91,1] = PR[GP1:90,1] + 33.098;
   1:  PR[GP1:91,2] = PR[GP1:90,2] + 15.735;
   1:L PR[91] R[100]mm/sec CNT100;
   1:  PR[GP1:91,1] = PR[GP1:90,1] + 28.739;
   1:  PR[GP1:91,2] = PR[GP1:90,2] + 17.686;
   1:L PR[91] R[100]mm/sec CNT100;
   1:  PR[GP1:91,1] = PR[GP1:90,1] + 28.081;
   1:  PR[GP1:91,2] = PR[GP1:90,2] + 17.921;
   1:L PR[91] R[100]mm/sec CNT100;
   1:  PR[GP1:91,1] = PR[GP1:90,1] + 27.400;
   1:  PR[GP1:91,2] = PR[GP1:90,2] + 18.044;
   1:L PR[91] R[100]mm/sec CNT100;
   1:  PR[GP1:91,1] = PR[GP1:90,1] + 22.645;
   1:  PR[GP1:91,2] = PR[GP1:90,2] + 18.485;
   1:L PR[91] R[100]mm/sec CNT100;
   1:  PR[GP1:91,1] = PR[GP1:90,1] + 21.946;
   1:  PR[GP1:91,2] = PR[GP1:90,2] + 18.496;
   1:L PR[91] R[100]mm/sec CNT100;
   1:  PR[GP1:91,1] = PR[GP1:90,1] + 21.262;
   1:  PR[GP1:91,2] = PR[GP1:90,2] + 18.394;
   1:L PR[91] R[100]mm/sec CNT100;
   1:  PR[GP1:91,1] = PR[GP1:90,1] + 16.619;
   1:  PR[GP1:91,2] = PR[GP1:90,2] + 17.276;
   1:L PR[91] R[100]mm/sec CNT100;
   1:  PR[GP1:91,1] = PR[GP1:90,1] + 15.953;
   1:  PR[GP1:91,2] = PR[GP1:90,2] + 17.062;
   1:L PR[91] R[100]mm/sec CNT100;
   1:  PR[GP1:91,1] = PR[GP1:90,1] + 15.339;
   1:  PR[GP1:91,2] = PR[GP1:90,2] + 16.746;
   1:L PR[91] R[100]mm/sec CNT100;
   1:  PR[GP1:91,1] = PR[GP1:90,1] + 11.306;
   1:  PR[GP1:91,2] = PR[GP1:90,2] + 14.190;
   1:L PR[91] R[100]mm/sec CNT100;
   1:  PR[GP1:91,1] = PR[GP1:90,1] + 10.743;
   1:  PR[GP1:91,2] = PR[GP1:90,2] + 13.772;
   1:L PR[91] R[100]mm/sec CNT100;
   1:  PR[GP1:91,1] = PR[GP1:90,1] + 10.264;
   1:  PR[GP1:91,2] = PR[GP1:90,2] + 13.276;
   1:L PR[91] R[100]mm/sec CNT100;
   1:  PR[GP1:91,1] = PR[GP1:90,1] + 7.270;
   1:  PR[GP1:91,2] = PR[GP1:90,2] + 9.557;
   1:L PR[91] R[100]mm/sec CNT100;
   1:  PR[GP1:91,1] = PR[GP1:90,1] + 6.871;
   1:  PR[GP1:91,2] = PR[GP1:90,2] + 8.979;
   1:L PR[91] R[100]mm/sec CNT100;
   1:  PR[GP1:91,1] = PR[GP1:90,1] + 6.578;
   1:  PR[GP1:91,2] = PR[GP1:90,2] + 8.356;
   1:L PR[91] R[100]mm/sec CNT100;
   1:  PR[GP1:91,1] = PR[GP1:90,1] + 4.947;
   1:  PR[GP1:91,2] = PR[GP1:90,2] + 3.878;
   1:L PR[91] R[100]mm/sec CNT100;
   1:  PR[GP1:91,1] = PR[GP1:90,1] + 4.688;
   1:  PR[GP1:91,2] = PR[GP1:90,2] + 2.953;
   1:L PR[91] R[100]mm/sec CNT100;
   1:  PR[GP1:91,1] = PR[GP1:90,1] + 4.285;
   1:  PR[GP1:91,2] = PR[GP1:90,2] + 1.996;
   1:L PR[91] R[100]mm/sec CNT100;
   1:  PR[GP1:91,1] = PR[GP1:90,1] + 3.919;
   1:  PR[GP1:91,2] = PR[GP1:90,2] + 1.565;
   1:L PR[91] R[100]mm/sec CNT100;
   1:  PR[GP1:91,1] = PR[GP1:90,1] + 3.337;
   1:  PR[GP1:91,2] = PR[GP1:90,2] + 1.083;
   1:L PR[91] R[100]mm/sec CNT100;
   1:  PR[GP1:91,1] = PR[GP1:90,1] + 2.846;
   1:  PR[GP1:91,2] = PR[GP1:90,2] + 0.801;
   1:L PR[91] R[100]mm/sec CNT100;
   1:  PR[GP1:91,1] = PR[GP1:90,1] + 1.770;
   1:  PR[GP1:91,2] = PR[GP1:90,2] + 0.568;
   1:L PR[91] R[100]mm/sec CNT100;
   1:  PR[GP1:91,1] = PR[GP1:90,1] + -1.613;
   1:L PR[91] R[100]mm/sec CNT100;
   1:  PR[91] = PR[90];
   1:  PR[GP1:91,1] = PR[GP1:90,1] + -2.649;
   1:  PR[GP1:91,2] = PR[GP1:90,2] + 0.783;
   1:  PR[GP1:91,3] = PR[GP1:90,3] + 2.135;
   1:L PR[91] R[100]mm/sec CNT100;
   1:  PR[GP1:91,1] = PR[GP1:90,1] + -3.242;
   1:  PR[GP1:91,2] = PR[GP1:90,2] + 1.123;
   1:L PR[91] R[100]mm/sec CNT100;
   1:  PR[GP1:91,1] = PR[GP1:90,1] + -3.711;
   1:  PR[GP1:91,2] = PR[GP1:90,2] + 1.512;
   1:L PR[91] R[100]mm/sec CNT100;
   1:  PR[GP1:91,1] = PR[GP1:90,1] + -4.141;
   1:  PR[GP1:91,2] = PR[GP1:90,2] + 2.017;
   1:L PR[91] R[100]mm/sec CNT100;
   1:  PR[GP1:91,1] = PR[GP1:90,1] + -4.390;
   1:  PR[GP1:91,2] = PR[GP1:90,2] + 2.581;
   1:L PR[91] R[100]mm/sec CNT100;
   1:  PR[GP1:91,1] = PR[GP1:90,1] + -5.550;
   1:  PR[GP1:91,2] = PR[GP1:90,2] + 5.756;
   1:L PR[91] R[100]mm/sec CNT100;
   1:  PR[GP1:91,1] = PR[GP1:90,1] + -5.931;
   1:  PR[GP1:91,2] = PR[GP1:90,2] + 6.842;
   1:L PR[91] R[100]mm/sec CNT100;
   1:  PR[GP1:91,1] = PR[GP1:90,1] + -6.269;
   1:  PR[GP1:91,2] = PR[GP1:90,2] + 8.030;
   1:L PR[91] R[100]mm/sec CNT100;
   1:  PR[GP1:91,1] = PR[GP1:90,1] + -6.704;
   1:  PR[GP1:91,2] = PR[GP1:90,2] + 8.952;
   1:L PR[91] R[100]mm/sec CNT100;
   1:  PR[GP1:91,1] = PR[GP1:90,1] + -9.150;
   1:  PR[GP1:91,2] = PR[GP1:90,2] + 11.992;
   1:L PR[91] R[100]mm/sec CNT100;
   1:  PR[GP1:91,1] = PR[GP1:90,1] + -9.857;
   1:  PR[GP1:91,2] = PR[GP1:90,2] + 13.015;
   1:L PR[91] R[100]mm/sec CNT100;
   1:  PR[GP1:91,1] = PR[GP1:90,1] + -10.565;
   1:  PR[GP1:91,2] = PR[GP1:90,2] + 13.748;
   1:L PR[91] R[100]mm/sec CNT100;
   1:  PR[GP1:91,1] = PR[GP1:90,1] + -13.861;
   1:  PR[GP1:91,2] = PR[GP1:90,2] + 15.836;
   1:L PR[91] R[100]mm/sec CNT100;
   1:  PR[GP1:91,1] = PR[GP1:90,1] + -14.859;
   1:  PR[GP1:91,2] = PR[GP1:90,2] + 16.578;
   1:L PR[91] R[100]mm/sec CNT100;
   1:  PR[GP1:91,1] = PR[GP1:90,1] + -15.765;
   1:  PR[GP1:91,2] = PR[GP1:90,2] + 17.044;
   1:L PR[91] R[100]mm/sec CNT100;
   1:  PR[GP1:91,1] = PR[GP1:90,1] + -19.558;
   1:  PR[GP1:91,2] = PR[GP1:90,2] + 17.957;
   1:L PR[91] R[100]mm/sec CNT100;
   1:  PR[GP1:91,1] = PR[GP1:90,1] + -20.743;
   1:  PR[GP1:91,2] = PR[GP1:90,2] + 18.339;
   1:L PR[91] R[100]mm/sec CNT100;
   1:  PR[GP1:91,1] = PR[GP1:90,1] + -21.749;
   1:  PR[GP1:91,2] = PR[GP1:90,2] + 18.489;
   1:L PR[91] R[100]mm/sec CNT100;
   1:  PR[GP1:91,1] = PR[GP1:90,1] + -25.635;
   1:  PR[GP1:91,2] = PR[GP1:90,2] + 18.129;
   1:L PR[91] R[100]mm/sec CNT100;
   1:  PR[GP1:91,1] = PR[GP1:90,1] + -26.881;
   1:  PR[GP1:91,2] = PR[GP1:90,2] + 18.109;
   1:L PR[91] R[100]mm/sec CNT100;
   1:  PR[GP1:91,1] = PR[GP1:90,1] + -27.881;
   1:  PR[GP1:91,2] = PR[GP1:90,2] + 17.928;
   1:L PR[91] R[100]mm/sec CNT100;
   1:  PR[GP1:91,1] = PR[GP1:90,1] + -31.443;
   1:  PR[GP1:91,2] = PR[GP1:90,2] + 16.334;
   1:L PR[91] R[100]mm/sec CNT100;
   1:  PR[GP1:91,1] = PR[GP1:90,1] + -32.617;
   1:  PR[GP1:91,2] = PR[GP1:90,2] + 15.914;
   1:L PR[91] R[100]mm/sec CNT100;
   1:  PR[GP1:91,1] = PR[GP1:90,1] + -33.505;
   1:  PR[GP1:91,2] = PR[GP1:90,2] + 15.421;
   1:L PR[91] R[100]mm/sec CNT100;
   1:  PR[GP1:91,1] = PR[GP1:90,1] + -36.361;
   1:  PR[GP1:91,2] = PR[GP1:90,2] + 12.763;
   1:L PR[91] R[100]mm/sec CNT100;
   1:  PR[GP1:91,1] = PR[GP1:90,1] + -37.339;
   1:  PR[GP1:91,2] = PR[GP1:90,2] + 11.988;
   1:L PR[91] R[100]mm/sec CNT100;
   1:  PR[GP1:91,1] = PR[GP1:90,1] + -38.021;
   1:  PR[GP1:91,2] = PR[GP1:90,2] + 11.236;
   1:L PR[91] R[100]mm/sec CNT100;
   1:  PR[GP1:91,1] = PR[GP1:90,1] + -39.867;
   1:  PR[GP1:91,2] = PR[GP1:90,2] + 7.798;
   1:L PR[91] R[100]mm/sec CNT100;
   1:  PR[GP1:91,1] = PR[GP1:90,1] + -40.544;
   1:  PR[GP1:91,2] = PR[GP1:90,2] + 6.749;
   1:L PR[91] R[100]mm/sec CNT100;
   1:  PR[GP1:91,1] = PR[GP1:90,1] + -40.947;
   1:  PR[GP1:91,2] = PR[GP1:90,2] + 5.819;
   1:L PR[91] R[100]mm/sec CNT100;
   1:  PR[GP1:91,1] = PR[GP1:90,1] + -41.585;
   1:  PR[GP1:91,2] = PR[GP1:90,2] + 1.969;
   1:L PR[91] R[100]mm/sec CNT100;
   1:  PR[GP1:91,1] = PR[GP1:90,1] + -41.889;
   1:  PR[GP1:91,2] = PR[GP1:90,2] + 0.757;
   1:L PR[91] R[100]mm/sec CNT100;
   1:  PR[GP1:91,1] = PR[GP1:90,1] + -41.972;
   1:  PR[GP1:91,2] = PR[GP1:90,2] + -0.252;
   1:L PR[91] R[100]mm/sec CNT100;
   1:  PR[GP1:91,1] = PR[GP1:90,1] + -41.334;
   1:  PR[GP1:91,2] = PR[GP1:90,2] + -4.102;
   1:L PR[91] R[100]mm/sec CNT100;
   1:  PR[GP1:91,1] = PR[GP1:90,1] + -41.231;
   1:  PR[GP1:91,2] = PR[GP1:90,2] + -5.348;
   1:L PR[91] R[100]mm/sec CNT100;
   1:  PR[GP1:91,1] = PR[GP1:90,1] + -40.971;
   1:  PR[GP1:91,2] = PR[GP1:90,2] + -6.389;
   1:L PR[91] R[100]mm/sec CNT100;
   1:  PR[GP1:91,1] = PR[GP1:90,1] + -40.521;
   1:  PR[GP1:91,2] = PR[GP1:90,2] + -7.426;
   1:L PR[91] R[100]mm/sec CNT100;
   1:  PR[GP1:91,1] = PR[GP1:90,1] + -38.674;
   1:  PR[GP1:91,2] = PR[GP1:90,2] + -10.865;
   1:L PR[91] R[100]mm/sec CNT100;
   1:  PR[GP1:91,1] = PR[GP1:90,1] + -38.060;
   1:  PR[GP1:91,2] = PR[GP1:90,2] + -11.817;
   1:L PR[91] R[100]mm/sec CNT100;
   1:  PR[GP1:91,1] = PR[GP1:90,1] + -37.301;
   1:  PR[GP1:91,2] = PR[GP1:90,2] + -12.654;
   1:L PR[91] R[100]mm/sec CNT100;
   1:  PR[GP1:91,1] = PR[GP1:90,1] + -34.443;
   1:  PR[GP1:91,2] = PR[GP1:90,2] + -15.313;
   1:L PR[91] R[100]mm/sec CNT100;
   1:  PR[GP1:91,1] = PR[GP1:90,1] + -33.555;
   1:  PR[GP1:91,2] = PR[GP1:90,2] + -16.017;
   1:L PR[91] R[100]mm/sec CNT100;
   1:  PR[GP1:91,1] = PR[GP1:90,1] + -32.568;
   1:  PR[GP1:91,2] = PR[GP1:90,2] + -16.565;
   1:L PR[91] R[100]mm/sec CNT100;
   1:  PR[GP1:91,1] = PR[GP1:90,1] + -29.005;
   1:  PR[GP1:91,2] = PR[GP1:90,2] + -18.160;
   1:L PR[91] R[100]mm/sec CNT100;
   1:  PR[GP1:91,1] = PR[GP1:90,1] + -27.936;
   1:  PR[GP1:91,2] = PR[GP1:90,2] + -18.542;
   1:L PR[91] R[100]mm/sec CNT100;
   1:  PR[GP1:91,1] = PR[GP1:90,1] + -26.826;
   1:  PR[GP1:91,2] = PR[GP1:90,2] + -18.743;
   1:L PR[91] R[100]mm/sec CNT100;
   1:  PR[GP1:91,1] = PR[GP1:90,1] + -22.940;
   1:  PR[GP1:91,2] = PR[GP1:90,2] + -19.103;
   1:L PR[91] R[100]mm/sec CNT100;
   1:  PR[GP1:91,1] = PR[GP1:90,1] + -21.805;
   1:  PR[GP1:91,2] = PR[GP1:90,2] + -19.121;
   1:L PR[91] R[100]mm/sec CNT100;
   1:  PR[GP1:91,1] = PR[GP1:90,1] + -20.689;
   1:  PR[GP1:91,2] = PR[GP1:90,2] + -18.955;
   1:L PR[91] R[100]mm/sec CNT100;
   1:  PR[GP1:91,1] = PR[GP1:90,1] + -16.895;
   1:  PR[GP1:91,2] = PR[GP1:90,2] + -18.041;
   1:L PR[91] R[100]mm/sec CNT100;
   1:  PR[GP1:91,1] = PR[GP1:90,1] + -15.813;
   1:  PR[GP1:91,2] = PR[GP1:90,2] + -17.693;
   1:L PR[91] R[100]mm/sec CNT100;
   1:  PR[GP1:91,1] = PR[GP1:90,1] + -14.812;
   1:  PR[GP1:91,2] = PR[GP1:90,2] + -17.177;
   1:L PR[91] R[100]mm/sec CNT100;
   1:  PR[GP1:91,1] = PR[GP1:90,1] + -11.515;
   1:  PR[GP1:91,2] = PR[GP1:90,2] + -15.089;
   1:L PR[91] R[100]mm/sec CNT100;
   1:  PR[GP1:91,1] = PR[GP1:90,1] + -10.602;
   1:  PR[GP1:91,2] = PR[GP1:90,2] + -14.411;
   1:L PR[91] R[100]mm/sec CNT100;
   1:  PR[GP1:91,1] = PR[GP1:90,1] + -9.820;
   1:  PR[GP1:91,2] = PR[GP1:90,2] + -13.601;
   1:L PR[91] R[100]mm/sec CNT100;
   1:  PR[GP1:91,1] = PR[GP1:90,1] + -7.374;
   1:  PR[GP1:91,2] = PR[GP1:90,2] + -10.561;
   1:L PR[91] R[100]mm/sec CNT100;
   1:  PR[GP1:91,1] = PR[GP1:90,1] + -6.727;
   1:  PR[GP1:91,2] = PR[GP1:90,2] + -9.624;
   1:L PR[91] R[100]mm/sec CNT100;
   1:  PR[GP1:91,1] = PR[GP1:90,1] + -6.247;
   1:  PR[GP1:91,2] = PR[GP1:90,2] + -8.607;
   1:L PR[91] R[100]mm/sec CNT100;
   1:  PR[GP1:91,1] = PR[GP1:90,1] + -4.914;
   1:  PR[GP1:91,2] = PR[GP1:90,2] + -4.948;
   1:L PR[91] R[100]mm/sec CNT100;
   1:  PR[GP1:91,1] = PR[GP1:90,1] + -4.533;
   1:  PR[GP1:91,2] = PR[GP1:90,2] + -3.584;
   1:L PR[91] R[100]mm/sec CNT100;
   1:  PR[GP1:91,1] = PR[GP1:90,1] + -4.154;
   1:  PR[GP1:91,2] = PR[GP1:90,2] + -2.656;
   1:L PR[91] R[100]mm/sec CNT100;
   1:  PR[GP1:91,1] = PR[GP1:90,1] + -3.711;
   1:  PR[GP1:91,2] = PR[GP1:90,2] + -2.136;
   1:L PR[91] R[100]mm/sec CNT100;
   1:  PR[GP1:91,1] = PR[GP1:90,1] + -3.242;
   1:  PR[GP1:91,2] = PR[GP1:90,2] + -1.746;
   1:L PR[91] R[100]mm/sec CNT100;
   1:  PR[GP1:91,1] = PR[GP1:90,1] + -2.649;
   1:  PR[GP1:91,2] = PR[GP1:90,2] + -1.407;
   1:L PR[91] R[100]mm/sec CNT100;
   1:  PR[GP1:91,1] = PR[GP1:90,1] + -1.606;
   1:  PR[GP1:91,2] = PR[GP1:90,2] + -1.192;
   1:L PR[91] R[100]mm/sec CNT100;
   1:  PR[GP1:91,1] = PR[GP1:90,1] + 1.763;
   1:L PR[91] R[100]mm/sec CNT100;
   1:  PR[GP1:91,1] = PR[GP1:90,1] + 2.806;
   1:  PR[GP1:91,2] = PR[GP1:90,2] + -1.407;
   1:L PR[91] R[100]mm/sec CNT100;
   1:  PR[GP1:91,1] = PR[GP1:90,1] + 3.399;
   1:  PR[GP1:91,2] = PR[GP1:90,2] + -1.746;
   1:L PR[91] R[100]mm/sec CNT100;
   1:  PR[GP1:91,1] = PR[GP1:90,1] + 3.868;
   1:  PR[GP1:91,2] = PR[GP1:90,2] + -2.136;
   1:L PR[91] R[100]mm/sec CNT100;
   1:  PR[GP1:91,1] = PR[GP1:90,1] + 4.311;
   1:  PR[GP1:91,2] = PR[GP1:90,2] + -2.656;
   1:L PR[91] R[100]mm/sec CNT100;
   1:  PR[GP1:91,1] = PR[GP1:90,1] + 4.669;
   1:  PR[GP1:91,2] = PR[GP1:90,2] + -3.533;
   1:L PR[91] R[100]mm/sec CNT100;
   1:  PR[GP1:91,1] = PR[GP1:90,1] + 5.901;
   1:  PR[GP1:91,2] = PR[GP1:90,2] + -6.922;
   1:L PR[91] R[100]mm/sec CNT100;
   1:  PR[GP1:91,1] = PR[GP1:90,1] + 6.090;
   1:  PR[GP1:91,2] = PR[GP1:90,2] + -7.471;
   1:L PR[91] R[100]mm/sec CNT100;
   1:  PR[GP1:91,1] = PR[GP1:90,1] + 6.426;
   1:  PR[GP1:91,2] = PR[GP1:90,2] + -8.654;
   1:L PR[91] R[100]mm/sec CNT100;
   1:  PR[GP1:91,1] = PR[GP1:90,1] + 6.861;
   1:  PR[GP1:91,2] = PR[GP1:90,2] + -9.576;
   1:L PR[91] R[100]mm/sec CNT100;
   1:  PR[GP1:91,1] = PR[GP1:90,1] + 9.307;
   1:  PR[GP1:91,2] = PR[GP1:90,2] + -12.616;
   1:L PR[91] R[100]mm/sec CNT100;
   1:  PR[GP1:91,1] = PR[GP1:90,1] + 10.014;
   1:  PR[GP1:91,2] = PR[GP1:90,2] + -13.639;
   1:L PR[91] R[100]mm/sec CNT100;
   1:  PR[GP1:91,1] = PR[GP1:90,1] + 10.721;
   1:  PR[GP1:91,2] = PR[GP1:90,2] + -14.372;
   1:L PR[91] R[100]mm/sec CNT100;
   1:  PR[GP1:91,1] = PR[GP1:90,1] + 14.017;
   1:  PR[GP1:91,2] = PR[GP1:90,2] + -16.460;
   1:L PR[91] R[100]mm/sec CNT100;
   1:  PR[GP1:91,1] = PR[GP1:90,1] + 15.016;
   1:  PR[GP1:91,2] = PR[GP1:90,2] + -17.202;
   1:L PR[91] R[100]mm/sec CNT100;
   1:  PR[GP1:91,1] = PR[GP1:90,1] + 15.921;
   1:  PR[GP1:91,2] = PR[GP1:90,2] + -17.668;
   1:L PR[91] R[100]mm/sec CNT100;
   1:  PR[GP1:91,1] = PR[GP1:90,1] + 19.715;
   1:  PR[GP1:91,2] = PR[GP1:90,2] + -18.581;
   1:L PR[91] R[100]mm/sec CNT100;
   1:  PR[GP1:91,1] = PR[GP1:90,1] + 20.900;
   1:  PR[GP1:91,2] = PR[GP1:90,2] + -18.963;
   1:L PR[91] R[100]mm/sec CNT100;
   1:  PR[GP1:91,1] = PR[GP1:90,1] + 21.906;
   1:  PR[GP1:91,2] = PR[GP1:90,2] + -19.113;
   1:L PR[91] R[100]mm/sec CNT100;
   1:  PR[GP1:91,1] = PR[GP1:90,1] + 25.792;
   1:  PR[GP1:91,2] = PR[GP1:90,2] + -18.753;
   1:L PR[91] R[100]mm/sec CNT100;
   1:  PR[GP1:91,1] = PR[GP1:90,1] + 27.038;
   1:  PR[GP1:91,2] = PR[GP1:90,2] + -18.733;
   1:L PR[91] R[100]mm/sec CNT100;
   1:  PR[GP1:91,1] = PR[GP1:90,1] + 28.038;
   1:  PR[GP1:91,2] = PR[GP1:90,2] + -18.552;
   1:L PR[91] R[100]mm/sec CNT100;
   1:  PR[GP1:91,1] = PR[GP1:90,1] + 31.599;
   1:  PR[GP1:91,2] = PR[GP1:90,2] + -16.958;
   1:L PR[91] R[100]mm/sec CNT100;
   1:  PR[GP1:91,1] = PR[GP1:90,1] + 32.774;
   1:  PR[GP1:91,2] = PR[GP1:90,2] + -16.538;
   1:L PR[91] R[100]mm/sec CNT100;
   1:  PR[GP1:91,1] = PR[GP1:90,1] + 33.661;
   1:  PR[GP1:91,2] = PR[GP1:90,2] + -16.045;
   1:L PR[91] R[100]mm/sec CNT100;
   1:  PR[GP1:91,1] = PR[GP1:90,1] + 36.518;
   1:  PR[GP1:91,2] = PR[GP1:90,2] + -13.387;
   1:L PR[91] R[100]mm/sec CNT100;
   1:  PR[GP1:91,1] = PR[GP1:90,1] + 37.496;
   1:  PR[GP1:91,2] = PR[GP1:90,2] + -12.612;
   1:L PR[91] R[100]mm/sec CNT100;
   1:  PR[GP1:91,1] = PR[GP1:90,1] + 38.177;
   1:  PR[GP1:91,2] = PR[GP1:90,2] + -11.860;
   1:L PR[91] R[100]mm/sec CNT100;
   1:  PR[GP1:91,1] = PR[GP1:90,1] + 40.024;
   1:  PR[GP1:91,2] = PR[GP1:90,2] + -8.422;
   1:L PR[91] R[100]mm/sec CNT100;
   1:  PR[GP1:91,1] = PR[GP1:90,1] + 40.701;
   1:  PR[GP1:91,2] = PR[GP1:90,2] + -7.373;
   1:L PR[91] R[100]mm/sec CNT100;
   1:  PR[GP1:91,1] = PR[GP1:90,1] + 41.104;
   1:  PR[GP1:91,2] = PR[GP1:90,2] + -6.443;
   1:L PR[91] R[100]mm/sec CNT100;
   1:  PR[GP1:91,1] = PR[GP1:90,1] + 41.742;
   1:  PR[GP1:91,2] = PR[GP1:90,2] + -2.593;
   1:L PR[91] R[100]mm/sec CNT100;
   1:  PR[GP1:91,1] = PR[GP1:90,1] + 42.046;
   1:  PR[GP1:91,2] = PR[GP1:90,2] + -1.381;
   1:L PR[91] R[100]mm/sec CNT100;
   1:  PR[GP1:91,1] = PR[GP1:90,1] + 42.129;
   1:  PR[GP1:91,2] = PR[GP1:90,2] + -0.372;
   1:L PR[91] R[100]mm/sec CNT100;
   1:  PR[GP1:91,1] = PR[GP1:90,1] + 41.490;
   1:  PR[GP1:91,2] = PR[GP1:90,2] + 3.478;
   1:L PR[91] R[100]mm/sec CNT100;
   1:  PR[GP1:91,1] = PR[GP1:90,1] + 41.388;
   1:  PR[GP1:91,2] = PR[GP1:90,2] + 4.724;
   1:L PR[91] R[100]mm/sec CNT100;
   1:  PR[GP1:91,1] = PR[GP1:90,1] + 41.127;
   1:  PR[GP1:91,2] = PR[GP1:90,2] + 5.765;
   1:L PR[91] R[100]mm/sec CNT100;
   1:  PR[GP1:91,1] = PR[GP1:90,1] + 40.678;
   1:  PR[GP1:91,2] = PR[GP1:90,2] + 6.802;
   1:L PR[91] R[100]mm/sec CNT100;
   1:  PR[GP1:91,1] = PR[GP1:90,1] + 38.831;
   1:  PR[GP1:91,2] = PR[GP1:90,2] + 10.241;
   1:L PR[91] R[100]mm/sec CNT100;
   1:  PR[GP1:91,1] = PR[GP1:90,1] + 38.217;
   1:  PR[GP1:91,2] = PR[GP1:90,2] + 11.193;
   1:L PR[91] R[100]mm/sec CNT100;
   1:  PR[GP1:91,1] = PR[GP1:90,1] + 37.458;
   1:  PR[GP1:91,2] = PR[GP1:90,2] + 12.030;
   1:L PR[91] R[100]mm/sec CNT100;
   1:  PR[GP1:91,1] = PR[GP1:90,1] + 34.600;
   1:  PR[GP1:91,2] = PR[GP1:90,2] + 14.689;
   1:L PR[91] R[100]mm/sec CNT100;
   1:  PR[GP1:91,1] = PR[GP1:90,1] + 33.712;
   1:  PR[GP1:91,2] = PR[GP1:90,2] + 15.393;
   1:L PR[91] R[100]mm/sec CNT100;
   1:  PR[GP1:91,1] = PR[GP1:90,1] + 32.724;
   1:  PR[GP1:91,2] = PR[GP1:90,2] + 15.941;
   1:L PR[91] R[100]mm/sec CNT100;
   1:  PR[GP1:91,1] = PR[GP1:90,1] + 29.162;
   1:  PR[GP1:91,2] = PR[GP1:90,2] + 17.536;
   1:L PR[91] R[100]mm/sec CNT100;
   1:  PR[GP1:91,1] = PR[GP1:90,1] + 28.093;
   1:  PR[GP1:91,2] = PR[GP1:90,2] + 17.918;
   1:L PR[91] R[100]mm/sec CNT100;
   1:  PR[GP1:91,1] = PR[GP1:90,1] + 26.983;
   1:  PR[GP1:91,2] = PR[GP1:90,2] + 18.119;
   1:L PR[91] R[100]mm/sec CNT100;
   1:  PR[GP1:91,1] = PR[GP1:90,1] + 23.097;
   1:  PR[GP1:91,2] = PR[GP1:90,2] + 18.479;
   1:L PR[91] R[100]mm/sec CNT100;
   1:  PR[GP1:91,1] = PR[GP1:90,1] + 21.961;
   1:  PR[GP1:91,2] = PR[GP1:90,2] + 18.497;
   1:L PR[91] R[100]mm/sec CNT100;
   1:  PR[GP1:91,1] = PR[GP1:90,1] + 20.846;
   1:  PR[GP1:91,2] = PR[GP1:90,2] + 18.331;
   1:L PR[91] R[100]mm/sec CNT100;
   1:  PR[GP1:91,1] = PR[GP1:90,1] + 17.052;
   1:  PR[GP1:91,2] = PR[GP1:90,2] + 17.417;
   1:L PR[91] R[100]mm/sec CNT100;
   1:  PR[GP1:91,1] = PR[GP1:90,1] + 15.970;
   1:  PR[GP1:91,2] = PR[GP1:90,2] + 17.069;
   1:L PR[91] R[100]mm/sec CNT100;
   1:  PR[GP1:91,1] = PR[GP1:90,1] + 14.968;
   1:  PR[GP1:91,2] = PR[GP1:90,2] + 16.553;
   1:L PR[91] R[100]mm/sec CNT100;
   1:  PR[GP1:91,1] = PR[GP1:90,1] + 11.672;
   1:  PR[GP1:91,2] = PR[GP1:90,2] + 14.465;
   1:L PR[91] R[100]mm/sec CNT100;
   1:  PR[GP1:91,1] = PR[GP1:90,1] + 10.759;
   1:  PR[GP1:91,2] = PR[GP1:90,2] + 13.787;
   1:L PR[91] R[100]mm/sec CNT100;
   1:  PR[GP1:91,1] = PR[GP1:90,1] + 9.977;
   1:  PR[GP1:91,2] = PR[GP1:90,2] + 12.977;
   1:L PR[91] R[100]mm/sec CNT100;
   1:  PR[GP1:91,1] = PR[GP1:90,1] + 7.530;
   1:  PR[GP1:91,2] = PR[GP1:90,2] + 9.937;
   1:L PR[91] R[100]mm/sec CNT100;
   1:  PR[GP1:91,1] = PR[GP1:90,1] + 6.884;
   1:  PR[GP1:91,2] = PR[GP1:90,2] + 9.000;
   1:L PR[91] R[100]mm/sec CNT100;
   1:  PR[GP1:91,1] = PR[GP1:90,1] + 6.404;
   1:  PR[GP1:91,2] = PR[GP1:90,2] + 7.983;
   1:L PR[91] R[100]mm/sec CNT100;
   1:  PR[GP1:91,1] = PR[GP1:90,1] + 5.071;
   1:  PR[GP1:91,2] = PR[GP1:90,2] + 4.324;
   1:L PR[91] R[100]mm/sec CNT100;
   1:  PR[GP1:91,1] = PR[GP1:90,1] + 4.690;
   1:  PR[GP1:91,2] = PR[GP1:90,2] + 2.960;
   1:L PR[91] R[100]mm/sec CNT100;
   1:  PR[GP1:91,1] = PR[GP1:90,1] + 4.311;
   1:  PR[GP1:91,2] = PR[GP1:90,2] + 2.032;
   1:L PR[91] R[100]mm/sec CNT100;
   1:  PR[GP1:91,1] = PR[GP1:90,1] + 3.868;
   1:  PR[GP1:91,2] = PR[GP1:90,2] + 1.512;
   1:L PR[91] R[100]mm/sec CNT100;
   1:  PR[GP1:91,1] = PR[GP1:90,1] + 3.399;
   1:  PR[GP1:91,2] = PR[GP1:90,2] + 1.123;
   1:L PR[91] R[100]mm/sec CNT100;
   1:  PR[GP1:91,1] = PR[GP1:90,1] + 2.806;
   1:  PR[GP1:91,2] = PR[GP1:90,2] + 0.783;
   1:L PR[91] R[100]mm/sec CNT100;
   1:  PR[GP1:91,1] = PR[GP1:90,1] + 1.763;
   1:  PR[GP1:91,2] = PR[GP1:90,2] + 0.568;
   1:L PR[91] R[100]mm/sec CNT100;
   1:  PR[GP1:91,1] = PR[GP1:90,1] + -1.606;
   1:L PR[91] R[100]mm/sec CNT100;
   1:  PR[91] = PR[90];
   1:  PR[GP1:91,1] = PR[GP1:90,1] + -2.608;
   1:  PR[GP1:91,2] = PR[GP1:90,2] + 0.765;
   1:  PR[GP1:91,3] = PR[GP1:90,3] + 2.745;
   1:L PR[91] R[100]mm/sec CNT100;
   1:  PR[GP1:91,1] = PR[GP1:90,1] + -3.303;
   1:  PR[GP1:91,2] = PR[GP1:90,2] + 1.162;
   1:L PR[91] R[100]mm/sec CNT100;
   1:  PR[GP1:91,1] = PR[GP1:90,1] + -3.661;
   1:  PR[GP1:91,2] = PR[GP1:90,2] + 1.459;
   1:L PR[91] R[100]mm/sec CNT100;
   1:  PR[GP1:91,1] = PR[GP1:90,1] + -4.180;
   1:  PR[GP1:91,2] = PR[GP1:90,2] + 2.069;
   1:L PR[91] R[100]mm/sec CNT100;
   1:  PR[GP1:91,1] = PR[GP1:90,1] + -4.516;
   1:  PR[GP1:91,2] = PR[GP1:90,2] + 2.919;
   1:L PR[91] R[100]mm/sec CNT100;
   1:  PR[GP1:91,1] = PR[GP1:90,1] + -5.637;
   1:  PR[GP1:91,2] = PR[GP1:90,2] + 6.045;
   1:L PR[91] R[100]mm/sec CNT100;
   1:  PR[GP1:91,1] = PR[GP1:90,1] + -6.095;
   1:  PR[GP1:91,2] = PR[GP1:90,2] + 7.657;
   1:L PR[91] R[100]mm/sec CNT100;
   1:  PR[GP1:91,1] = PR[GP1:90,1] + -6.716;
   1:  PR[GP1:91,2] = PR[GP1:90,2] + 8.974;
   1:L PR[91] R[100]mm/sec CNT100;
   1:  PR[GP1:91,1] = PR[GP1:90,1] + -8.615;
   1:  PR[GP1:91,2] = PR[GP1:90,2] + 11.333;
   1:L PR[91] R[100]mm/sec CNT100;
   1:  PR[GP1:91,1] = PR[GP1:90,1] + -9.570;
   1:  PR[GP1:91,2] = PR[GP1:90,2] + 12.716;
   1:L PR[91] R[100]mm/sec CNT100;
   1:  PR[GP1:91,1] = PR[GP1:90,1] + -10.581;
   1:  PR[GP1:91,2] = PR[GP1:90,2] + 13.762;
   1:L PR[91] R[100]mm/sec CNT100;
   1:  PR[GP1:91,1] = PR[GP1:90,1] + -13.139;
   1:  PR[GP1:91,2] = PR[GP1:90,2] + 15.383;
   1:L PR[91] R[100]mm/sec CNT100;
   1:  PR[GP1:91,1] = PR[GP1:90,1] + -14.489;
   1:  PR[GP1:91,2] = PR[GP1:90,2] + 16.386;
   1:L PR[91] R[100]mm/sec CNT100;
   1:  PR[GP1:91,1] = PR[GP1:90,1] + -15.782;
   1:  PR[GP1:91,2] = PR[GP1:90,2] + 17.051;
   1:L PR[91] R[100]mm/sec CNT100;
   1:  PR[GP1:91,1] = PR[GP1:90,1] + -18.727;
   1:  PR[GP1:91,2] = PR[GP1:90,2] + 17.760;
   1:L PR[91] R[100]mm/sec CNT100;
   1:  PR[GP1:91,1] = PR[GP1:90,1] + -20.327;
   1:  PR[GP1:91,2] = PR[GP1:90,2] + 18.276;
   1:L PR[91] R[100]mm/sec CNT100;
   1:  PR[GP1:91,1] = PR[GP1:90,1] + -21.765;
   1:  PR[GP1:91,2] = PR[GP1:90,2] + 18.490;
   1:L PR[91] R[100]mm/sec CNT100;
   1:  PR[GP1:91,1] = PR[GP1:90,1] + -24.781;
   1:  PR[GP1:91,2] = PR[GP1:90,2] + 18.210;
   1:L PR[91] R[100]mm/sec CNT100;
   1:  PR[GP1:91,1] = PR[GP1:90,1] + -26.464;
   1:  PR[GP1:91,2] = PR[GP1:90,2] + 18.184;
   1:L PR[91] R[100]mm/sec CNT100;
   1:  PR[GP1:91,1] = PR[GP1:90,1] + -27.893;
   1:  PR[GP1:91,2] = PR[GP1:90,2] + 17.925;
   1:L PR[91] R[100]mm/sec CNT100;
   1:  PR[GP1:91,1] = PR[GP1:90,1] + -30.658;
   1:  PR[GP1:91,2] = PR[GP1:90,2] + 16.687;
   1:L PR[91] R[100]mm/sec CNT100;
   1:  PR[GP1:91,1] = PR[GP1:90,1] + -32.243;
   1:  PR[GP1:91,2] = PR[GP1:90,2] + 16.121;
   1:L PR[91] R[100]mm/sec CNT100;
   1:  PR[GP1:91,1] = PR[GP1:90,1] + -33.512;
   1:  PR[GP1:91,2] = PR[GP1:90,2] + 15.416;
   1:L PR[91] R[100]mm/sec CNT100;
   1:  PR[GP1:91,1] = PR[GP1:90,1] + -35.730;
   1:  PR[GP1:91,2] = PR[GP1:90,2] + 13.352;
   1:L PR[91] R[100]mm/sec CNT100;
   1:  PR[GP1:91,1] = PR[GP1:90,1] + -37.050;
   1:  PR[GP1:91,2] = PR[GP1:90,2] + 12.306;
   1:L PR[91] R[100]mm/sec CNT100;
   1:  PR[GP1:91,1] = PR[GP1:90,1] + -38.025;
   1:  PR[GP1:91,2] = PR[GP1:90,2] + 11.231;
   1:L PR[91] R[100]mm/sec CNT100;
   1:  PR[GP1:91,1] = PR[GP1:90,1] + -39.458;
   1:  PR[GP1:91,2] = PR[GP1:90,2] + 8.562;
   1:L PR[91] R[100]mm/sec CNT100;
   1:  PR[GP1:91,1] = PR[GP1:90,1] + -40.371;
   1:  PR[GP1:91,2] = PR[GP1:90,2] + 7.146;
   1:L PR[91] R[100]mm/sec CNT100;
   1:  PR[GP1:91,1] = PR[GP1:90,1] + -40.948;
   1:  PR[GP1:91,2] = PR[GP1:90,2] + 5.816;
   1:L PR[91] R[100]mm/sec CNT100;
   1:  PR[GP1:91,1] = PR[GP1:90,1] + -41.444;
   1:  PR[GP1:91,2] = PR[GP1:90,2] + 2.827;
   1:L PR[91] R[100]mm/sec CNT100;
   1:  PR[GP1:91,1] = PR[GP1:90,1] + -41.853;
   1:  PR[GP1:91,2] = PR[GP1:90,2] + 1.192;
   1:L PR[91] R[100]mm/sec CNT100;
   1:  PR[GP1:91,1] = PR[GP1:90,1] + -41.972;
   1:  PR[GP1:91,2] = PR[GP1:90,2] + -0.252;
   1:L PR[91] R[100]mm/sec CNT100;
   1:  PR[GP1:91,1] = PR[GP1:90,1] + -41.476;
   1:  PR[GP1:91,2] = PR[GP1:90,2] + -3.241;
   1:L PR[91] R[100]mm/sec CNT100;
   1:  PR[GP1:91,1] = PR[GP1:90,1] + -41.339;
   1:  PR[GP1:91,2] = PR[GP1:90,2] + -4.922;
   1:L PR[91] R[100]mm/sec CNT100;
   1:  PR[GP1:91,1] = PR[GP1:90,1] + -40.972;
   1:  PR[GP1:91,2] = PR[GP1:90,2] + -6.386;
   1:L PR[91] R[100]mm/sec CNT100;
   1:  PR[GP1:91,1] = PR[GP1:90,1] + -40.348;
   1:  PR[GP1:91,2] = PR[GP1:90,2] + -7.823;
   1:L PR[91] R[100]mm/sec CNT100;
   1:  PR[GP1:91,1] = PR[GP1:90,1] + -38.915;
   1:  PR[GP1:91,2] = PR[GP1:90,2] + -10.493;
   1:L PR[91] R[100]mm/sec CNT100;
   1:  PR[GP1:91,1] = PR[GP1:90,1] + -38.064;
   1:  PR[GP1:91,2] = PR[GP1:90,2] + -11.812;
   1:L PR[91] R[100]mm/sec CNT100;
   1:  PR[GP1:91,1] = PR[GP1:90,1] + -37.011;
   1:  PR[GP1:91,2] = PR[GP1:90,2] + -12.972;
   1:L PR[91] R[100]mm/sec CNT100;
   1:  PR[GP1:91,1] = PR[GP1:90,1] + -34.793;
   1:  PR[GP1:91,2] = PR[GP1:90,2] + -15.036;
   1:L PR[91] R[100]mm/sec CNT100;
   1:  PR[GP1:91,1] = PR[GP1:90,1] + -33.563;
   1:  PR[GP1:91,2] = PR[GP1:90,2] + -16.012;
   1:L PR[91] R[100]mm/sec CNT100;
   1:  PR[GP1:91,1] = PR[GP1:90,1] + -32.194;
   1:  PR[GP1:91,2] = PR[GP1:90,2] + -16.772;
   1:L PR[91] R[100]mm/sec CNT100;
   1:  PR[GP1:91,1] = PR[GP1:90,1] + -29.428;
   1:  PR[GP1:91,2] = PR[GP1:90,2] + -18.010;
   1:L PR[91] R[100]mm/sec CNT100;
   1:  PR[GP1:91,1] = PR[GP1:90,1] + -27.949;
   1:  PR[GP1:91,2] = PR[GP1:90,2] + -18.539;
   1:L PR[91] R[100]mm/sec CNT100;
   1:  PR[GP1:91,1] = PR[GP1:90,1] + -26.409;
   1:  PR[GP1:91,2] = PR[GP1:90,2] + -18.818;
   1:L PR[91] R[100]mm/sec CNT100;
   1:  PR[GP1:91,1] = PR[GP1:90,1] + -23.392;
   1:  PR[GP1:91,2] = PR[GP1:90,2] + -19.097;
   1:L PR[91] R[100]mm/sec CNT100;
   1:  PR[GP1:91,1] = PR[GP1:90,1] + -21.820;
   1:  PR[GP1:91,2] = PR[GP1:90,2] + -19.122;
   1:L PR[91] R[100]mm/sec CNT100;
   1:  PR[GP1:91,1] = PR[GP1:90,1] + -20.273;
   1:  PR[GP1:91,2] = PR[GP1:90,2] + -18.891;
   1:L PR[91] R[100]mm/sec CNT100;
   1:  PR[GP1:91,1] = PR[GP1:90,1] + -17.328;
   1:  PR[GP1:91,2] = PR[GP1:90,2] + -18.182;
   1:L PR[91] R[100]mm/sec CNT100;
   1:  PR[GP1:91,1] = PR[GP1:90,1] + -15.831;
   1:  PR[GP1:91,2] = PR[GP1:90,2] + -17.700;
   1:L PR[91] R[100]mm/sec CNT100;
   1:  PR[GP1:91,1] = PR[GP1:90,1] + -14.441;
   1:  PR[GP1:91,2] = PR[GP1:90,2] + -16.985;
   1:L PR[91] R[100]mm/sec CNT100;
   1:  PR[GP1:91,1] = PR[GP1:90,1] + -11.882;
   1:  PR[GP1:91,2] = PR[GP1:90,2] + -15.364;
   1:L PR[91] R[100]mm/sec CNT100;
   1:  PR[GP1:91,1] = PR[GP1:90,1] + -10.618;
   1:  PR[GP1:91,2] = PR[GP1:90,2] + -14.425;
   1:L PR[91] R[100]mm/sec CNT100;
   1:  PR[GP1:91,1] = PR[GP1:90,1] + -9.533;
   1:  PR[GP1:91,2] = PR[GP1:90,2] + -13.301;
   1:L PR[91] R[100]mm/sec CNT100;
   1:  PR[GP1:91,1] = PR[GP1:90,1] + -7.634;
   1:  PR[GP1:91,2] = PR[GP1:90,2] + -10.941;
   1:L PR[91] R[100]mm/sec CNT100;
   1:  PR[GP1:91,1] = PR[GP1:90,1] + -6.739;
   1:  PR[GP1:91,2] = PR[GP1:90,2] + -9.646;
   1:L PR[91] R[100]mm/sec CNT100;
   1:  PR[GP1:91,1] = PR[GP1:90,1] + -6.073;
   1:  PR[GP1:91,2] = PR[GP1:90,2] + -8.233;
   1:L PR[91] R[100]mm/sec CNT100;
   1:  PR[GP1:91,1] = PR[GP1:90,1] + -5.038;
   1:  PR[GP1:91,2] = PR[GP1:90,2] + -5.394;
   1:L PR[91] R[100]mm/sec CNT100;
   1:  PR[GP1:91,1] = PR[GP1:90,1] + -4.536;
   1:  PR[GP1:91,2] = PR[GP1:90,2] + -3.591;
   1:L PR[91] R[100]mm/sec CNT100;
   1:  PR[GP1:91,1] = PR[GP1:90,1] + -4.180;
   1:  PR[GP1:91,2] = PR[GP1:90,2] + -2.693;
   1:L PR[91] R[100]mm/sec CNT100;
   1:  PR[GP1:91,1] = PR[GP1:90,1] + -3.661;
   1:  PR[GP1:91,2] = PR[GP1:90,2] + -2.083;
   1:L PR[91] R[100]mm/sec CNT100;
   1:  PR[GP1:91,1] = PR[GP1:90,1] + -3.303;
   1:  PR[GP1:91,2] = PR[GP1:90,2] + -1.786;
   1:L PR[91] R[100]mm/sec CNT100;
   1:  PR[GP1:91,1] = PR[GP1:90,1] + -2.608;
   1:  PR[GP1:91,2] = PR[GP1:90,2] + -1.389;
   1:L PR[91] R[100]mm/sec CNT100;
   1:  PR[GP1:91,1] = PR[GP1:90,1] + -1.598;
   1:  PR[GP1:91,2] = PR[GP1:90,2] + -1.192;
   1:L PR[91] R[100]mm/sec CNT100;
   1:  PR[GP1:91,1] = PR[GP1:90,1] + 1.754;
   1:L PR[91] R[100]mm/sec CNT100;
   1:  PR[GP1:91,1] = PR[GP1:90,1] + 2.765;
   1:  PR[GP1:91,2] = PR[GP1:90,2] + -1.389;
   1:L PR[91] R[100]mm/sec CNT100;
   1:  PR[GP1:91,1] = PR[GP1:90,1] + 3.460;
   1:  PR[GP1:91,2] = PR[GP1:90,2] + -1.786;
   1:L PR[91] R[100]mm/sec CNT100;
   1:  PR[GP1:91,1] = PR[GP1:90,1] + 3.817;
   1:  PR[GP1:91,2] = PR[GP1:90,2] + -2.083;
   1:L PR[91] R[100]mm/sec CNT100;
   1:  PR[GP1:91,1] = PR[GP1:90,1] + 4.336;
   1:  PR[GP1:91,2] = PR[GP1:90,2] + -2.693;
   1:L PR[91] R[100]mm/sec CNT100;
   1:  PR[GP1:91,1] = PR[GP1:90,1] + 4.673;
   1:  PR[GP1:91,2] = PR[GP1:90,2] + -3.543;
   1:L PR[91] R[100]mm/sec CNT100;
   1:  PR[GP1:91,1] = PR[GP1:90,1] + 5.794;
   1:  PR[GP1:91,2] = PR[GP1:90,2] + -6.669;
   1:L PR[91] R[100]mm/sec CNT100;
   1:  PR[GP1:91,1] = PR[GP1:90,1] + 6.252;
   1:  PR[GP1:91,2] = PR[GP1:90,2] + -8.281;
   1:L PR[91] R[100]mm/sec CNT100;
   1:  PR[GP1:91,1] = PR[GP1:90,1] + 6.873;
   1:  PR[GP1:91,2] = PR[GP1:90,2] + -9.598;
   1:L PR[91] R[100]mm/sec CNT100;
   1:  PR[GP1:91,1] = PR[GP1:90,1] + 8.772;
   1:  PR[GP1:91,2] = PR[GP1:90,2] + -11.957;
   1:L PR[91] R[100]mm/sec CNT100;
   1:  PR[GP1:91,1] = PR[GP1:90,1] + 9.727;
   1:  PR[GP1:91,2] = PR[GP1:90,2] + -13.340;
   1:L PR[91] R[100]mm/sec CNT100;
   1:  PR[GP1:91,1] = PR[GP1:90,1] + 10.738;
   1:  PR[GP1:91,2] = PR[GP1:90,2] + -14.386;
   1:L PR[91] R[100]mm/sec CNT100;
   1:  PR[GP1:91,1] = PR[GP1:90,1] + 13.296;
   1:  PR[GP1:91,2] = PR[GP1:90,2] + -16.007;
   1:L PR[91] R[100]mm/sec CNT100;
   1:  PR[GP1:91,1] = PR[GP1:90,1] + 14.645;
   1:  PR[GP1:91,2] = PR[GP1:90,2] + -17.009;
   1:L PR[91] R[100]mm/sec CNT100;
   1:  PR[GP1:91,1] = PR[GP1:90,1] + 15.939;
   1:  PR[GP1:91,2] = PR[GP1:90,2] + -17.675;
   1:L PR[91] R[100]mm/sec CNT100;
   1:  PR[GP1:91,1] = PR[GP1:90,1] + 18.884;
   1:  PR[GP1:91,2] = PR[GP1:90,2] + -18.384;
   1:L PR[91] R[100]mm/sec CNT100;
   1:  PR[GP1:91,1] = PR[GP1:90,1] + 20.484;
   1:  PR[GP1:91,2] = PR[GP1:90,2] + -18.899;
   1:L PR[91] R[100]mm/sec CNT100;
   1:  PR[GP1:91,1] = PR[GP1:90,1] + 21.922;
   1:  PR[GP1:91,2] = PR[GP1:90,2] + -19.114;
   1:L PR[91] R[100]mm/sec CNT100;
   1:  PR[GP1:91,1] = PR[GP1:90,1] + 24.938;
   1:  PR[GP1:91,2] = PR[GP1:90,2] + -18.834;
   1:L PR[91] R[100]mm/sec CNT100;
   1:  PR[GP1:91,1] = PR[GP1:90,1] + 26.620;
   1:  PR[GP1:91,2] = PR[GP1:90,2] + -18.808;
   1:L PR[91] R[100]mm/sec CNT100;
   1:  PR[GP1:91,1] = PR[GP1:90,1] + 28.050;
   1:  PR[GP1:91,2] = PR[GP1:90,2] + -18.549;
   1:L PR[91] R[100]mm/sec CNT100;
   1:  PR[GP1:91,1] = PR[GP1:90,1] + 30.815;
   1:  PR[GP1:91,2] = PR[GP1:90,2] + -17.311;
   1:L PR[91] R[100]mm/sec CNT100;
   1:  PR[GP1:91,1] = PR[GP1:90,1] + 32.400;
   1:  PR[GP1:91,2] = PR[GP1:90,2] + -16.745;
   1:L PR[91] R[100]mm/sec CNT100;
   1:  PR[GP1:91,1] = PR[GP1:90,1] + 33.669;
   1:  PR[GP1:91,2] = PR[GP1:90,2] + -16.040;
   1:L PR[91] R[100]mm/sec CNT100;
   1:  PR[GP1:91,1] = PR[GP1:90,1] + 35.887;
   1:  PR[GP1:91,2] = PR[GP1:90,2] + -13.976;
   1:L PR[91] R[100]mm/sec CNT100;
   1:  PR[GP1:91,1] = PR[GP1:90,1] + 37.207;
   1:  PR[GP1:91,2] = PR[GP1:90,2] + -12.930;
   1:L PR[91] R[100]mm/sec CNT100;
   1:  PR[GP1:91,1] = PR[GP1:90,1] + 38.181;
   1:  PR[GP1:91,2] = PR[GP1:90,2] + -11.855;
   1:L PR[91] R[100]mm/sec CNT100;
   1:  PR[GP1:91,1] = PR[GP1:90,1] + 39.615;
   1:  PR[GP1:91,2] = PR[GP1:90,2] + -9.186;
   1:L PR[91] R[100]mm/sec CNT100;
   1:  PR[GP1:91,1] = PR[GP1:90,1] + 40.528;
   1:  PR[GP1:91,2] = PR[GP1:90,2] + -7.770;
   1:L PR[91] R[100]mm/sec CNT100;
   1:  PR[GP1:91,1] = PR[GP1:90,1] + 41.105;
   1:  PR[GP1:91,2] = PR[GP1:90,2] + -6.440;
   1:L PR[91] R[100]mm/sec CNT100;
   1:  PR[GP1:91,1] = PR[GP1:90,1] + 41.600;
   1:  PR[GP1:91,2] = PR[GP1:90,2] + -3.451;
   1:L PR[91] R[100]mm/sec CNT100;
   1:  PR[GP1:91,1] = PR[GP1:90,1] + 42.010;
   1:  PR[GP1:91,2] = PR[GP1:90,2] + -1.816;
   1:L PR[91] R[100]mm/sec CNT100;
   1:  PR[GP1:91,1] = PR[GP1:90,1] + 42.129;
   1:  PR[GP1:91,2] = PR[GP1:90,2] + -0.372;
   1:L PR[91] R[100]mm/sec CNT100;
   1:  PR[GP1:91,1] = PR[GP1:90,1] + 41.633;
   1:  PR[GP1:91,2] = PR[GP1:90,2] + 2.617;
   1:L PR[91] R[100]mm/sec CNT100;
   1:  PR[GP1:91,1] = PR[GP1:90,1] + 41.495;
   1:  PR[GP1:91,2] = PR[GP1:90,2] + 4.298;
   1:L PR[91] R[100]mm/sec CNT100;
   1:  PR[GP1:91,1] = PR[GP1:90,1] + 41.128;
   1:  PR[GP1:91,2] = PR[GP1:90,2] + 5.762;
   1:L PR[91] R[100]mm/sec CNT100;
   1:  PR[GP1:91,1] = PR[GP1:90,1] + 40.505;
   1:  PR[GP1:91,2] = PR[GP1:90,2] + 7.199;
   1:L PR[91] R[100]mm/sec CNT100;
   1:  PR[GP1:91,1] = PR[GP1:90,1] + 39.071;
   1:  PR[GP1:91,2] = PR[GP1:90,2] + 9.869;
   1:L PR[91] R[100]mm/sec CNT100;
   1:  PR[GP1:91,1] = PR[GP1:90,1] + 38.220;
   1:  PR[GP1:91,2] = PR[GP1:90,2] + 11.188;
   1:L PR[91] R[100]mm/sec CNT100;
   1:  PR[GP1:91,1] = PR[GP1:90,1] + 37.168;
   1:  PR[GP1:91,2] = PR[GP1:90,2] + 12.348;
   1:L PR[91] R[100]mm/sec CNT100;
   1:  PR[GP1:91,1] = PR[GP1:90,1] + 34.950;
   1:  PR[GP1:91,2] = PR[GP1:90,2] + 14.412;
   1:L PR[91] R[100]mm/sec CNT100;
   1:  PR[GP1:91,1] = PR[GP1:90,1] + 33.719;
   1:  PR[GP1:91,2] = PR[GP1:90,2] + 15.388;
   1:L PR[91] R[100]mm/sec CNT100;
   1:  PR[GP1:91,1] = PR[GP1:90,1] + 32.351;
   1:  PR[GP1:91,2] = PR[GP1:90,2] + 16.148;
   1:L PR[91] R[100]mm/sec CNT100;
   1:  PR[GP1:91,1] = PR[GP1:90,1] + 29.585;
   1:  PR[GP1:91,2] = PR[GP1:90,2] + 17.386;
   1:L PR[91] R[100]mm/sec CNT100;
   1:  PR[GP1:91,1] = PR[GP1:90,1] + 28.105;
   1:  PR[GP1:91,2] = PR[GP1:90,2] + 17.915;
   1:L PR[91] R[100]mm/sec CNT100;
   1:  PR[GP1:91,1] = PR[GP1:90,1] + 26.566;
   1:  PR[GP1:91,2] = PR[GP1:90,2] + 18.194;
   1:L PR[91] R[100]mm/sec CNT100;
   1:  PR[GP1:91,1] = PR[GP1:90,1] + 23.549;
   1:  PR[GP1:91,2] = PR[GP1:90,2] + 18.473;
   1:L PR[91] R[100]mm/sec CNT100;
   1:  PR[GP1:91,1] = PR[GP1:90,1] + 21.977;
   1:  PR[GP1:91,2] = PR[GP1:90,2] + 18.498;
   1:L PR[91] R[100]mm/sec CNT100;
   1:  PR[GP1:91,1] = PR[GP1:90,1] + 20.430;
   1:  PR[GP1:91,2] = PR[GP1:90,2] + 18.267;
   1:L PR[91] R[100]mm/sec CNT100;
   1:  PR[GP1:91,1] = PR[GP1:90,1] + 17.484;
   1:  PR[GP1:91,2] = PR[GP1:90,2] + 17.558;
   1:L PR[91] R[100]mm/sec CNT100;
   1:  PR[GP1:91,1] = PR[GP1:90,1] + 15.987;
   1:  PR[GP1:91,2] = PR[GP1:90,2] + 17.076;
   1:L PR[91] R[100]mm/sec CNT100;
   1:  PR[GP1:91,1] = PR[GP1:90,1] + 14.598;
   1:  PR[GP1:91,2] = PR[GP1:90,2] + 16.361;
   1:L PR[91] R[100]mm/sec CNT100;
   1:  PR[GP1:91,1] = PR[GP1:90,1] + 12.038;
   1:  PR[GP1:91,2] = PR[GP1:90,2] + 14.740;
   1:L PR[91] R[100]mm/sec CNT100;
   1:  PR[GP1:91,1] = PR[GP1:90,1] + 10.775;
   1:  PR[GP1:91,2] = PR[GP1:90,2] + 13.801;
   1:L PR[91] R[100]mm/sec CNT100;
   1:  PR[GP1:91,1] = PR[GP1:90,1] + 9.690;
   1:  PR[GP1:91,2] = PR[GP1:90,2] + 12.677;
   1:L PR[91] R[100]mm/sec CNT100;
   1:  PR[GP1:91,1] = PR[GP1:90,1] + 7.790;
   1:  PR[GP1:91,2] = PR[GP1:90,2] + 10.317;
   1:L PR[91] R[100]mm/sec CNT100;
   1:  PR[GP1:91,1] = PR[GP1:90,1] + 6.896;
   1:  PR[GP1:91,2] = PR[GP1:90,2] + 9.022;
   1:L PR[91] R[100]mm/sec CNT100;
   1:  PR[GP1:91,1] = PR[GP1:90,1] + 6.230;
   1:  PR[GP1:91,2] = PR[GP1:90,2] + 7.609;
   1:L PR[91] R[100]mm/sec CNT100;
   1:  PR[GP1:91,1] = PR[GP1:90,1] + 5.195;
   1:  PR[GP1:91,2] = PR[GP1:90,2] + 4.770;
   1:L PR[91] R[100]mm/sec CNT100;
   1:  PR[GP1:91,1] = PR[GP1:90,1] + 4.692;
   1:  PR[GP1:91,2] = PR[GP1:90,2] + 2.967;
   1:L PR[91] R[100]mm/sec CNT100;
   1:  PR[GP1:91,1] = PR[GP1:90,1] + 4.336;
   1:  PR[GP1:91,2] = PR[GP1:90,2] + 2.069;
   1:L PR[91] R[100]mm/sec CNT100;
   1:  PR[GP1:91,1] = PR[GP1:90,1] + 3.817;
   1:  PR[GP1:91,2] = PR[GP1:90,2] + 1.459;
   1:L PR[91] R[100]mm/sec CNT100;
   1:  PR[GP1:91,1] = PR[GP1:90,1] + 3.460;
   1:  PR[GP1:91,2] = PR[GP1:90,2] + 1.162;
   1:L PR[91] R[100]mm/sec CNT100;
   1:  PR[GP1:91,1] = PR[GP1:90,1] + 2.765;
   1:  PR[GP1:91,2] = PR[GP1:90,2] + 0.765;
   1:L PR[91] R[100]mm/sec CNT100;
   1:  PR[GP1:91,1] = PR[GP1:90,1] + 1.754;
   1:  PR[GP1:91,2] = PR[GP1:90,2] + 0.568;
   1:L PR[91] R[100]mm/sec CNT100;
   1:  PR[GP1:91,1] = PR[GP1:90,1] + -1.598;
   1:L PR[91] R[100]mm/sec CNT100;
   1:  PR[91] = PR[90];
   1:  PR[GP1:91,1] = PR[GP1:90,1] + -2.566;
   1:  PR[GP1:91,2] = PR[GP1:90,2] + 0.746;
   1:  PR[GP1:91,3] = PR[GP1:90,3] + 3.355;
   1:L PR[91] R[100]mm/sec CNT100;
   1:  PR[GP1:91,1] = PR[GP1:90,1] + -3.365;
   1:  PR[GP1:91,2] = PR[GP1:90,2] + 1.202;
   1:L PR[91] R[100]mm/sec CNT100;
   1:  PR[GP1:91,1] = PR[GP1:90,1] + -3.610;
   1:  PR[GP1:91,2] = PR[GP1:90,2] + 1.406;
   1:L PR[91] R[100]mm/sec CNT100;
   1:  PR[GP1:91,1] = PR[GP1:90,1] + -4.210;
   1:  PR[GP1:91,2] = PR[GP1:90,2] + 2.111;
   1:L PR[91] R[100]mm/sec CNT100;
   1:  PR[GP1:91,1] = PR[GP1:90,1] + -4.719;
   1:  PR[GP1:91,2] = PR[GP1:90,2] + 3.474;
   1:L PR[91] R[100]mm/sec CNT100;
   1:  PR[GP1:91,1] = PR[GP1:90,1] + -5.345;
   1:  PR[GP1:91,2] = PR[GP1:90,2] + 5.256;
   1:L PR[91] R[100]mm/sec CNT100;
   1:  PR[GP1:91,1] = PR[GP1:90,1] + -5.921;
   1:  PR[GP1:91,2] = PR[GP1:90,2] + 7.283;
   1:L PR[91] R[100]mm/sec CNT100;
   1:  PR[GP1:91,1] = PR[GP1:90,1] + -6.728;
   1:  PR[GP1:91,2] = PR[GP1:90,2] + 8.995;
   1:L PR[91] R[100]mm/sec CNT100;
   1:  PR[GP1:91,1] = PR[GP1:90,1] + -8.080;
   1:  PR[GP1:91,2] = PR[GP1:90,2] + 10.675;
   1:L PR[91] R[100]mm/sec CNT100;
   1:  PR[GP1:91,1] = PR[GP1:90,1] + -9.283;
   1:  PR[GP1:91,2] = PR[GP1:90,2] + 12.416;
   1:L PR[91] R[100]mm/sec CNT100;
   1:  PR[GP1:91,1] = PR[GP1:90,1] + -10.597;
   1:  PR[GP1:91,2] = PR[GP1:90,2] + 13.776;
   1:L PR[91] R[100]mm/sec CNT100;
   1:  PR[GP1:91,1] = PR[GP1:90,1] + -12.418;
   1:  PR[GP1:91,2] = PR[GP1:90,2] + 14.930;
   1:L PR[91] R[100]mm/sec CNT100;
   1:  PR[GP1:91,1] = PR[GP1:90,1] + -14.118;
   1:  PR[GP1:91,2] = PR[GP1:90,2] + 16.193;
   1:L PR[91] R[100]mm/sec CNT100;
   1:  PR[GP1:91,1] = PR[GP1:90,1] + -15.799;
   1:  PR[GP1:91,2] = PR[GP1:90,2] + 17.058;
   1:L PR[91] R[100]mm/sec CNT100;
   1:  PR[GP1:91,1] = PR[GP1:90,1] + -17.895;
   1:  PR[GP1:91,2] = PR[GP1:90,2] + 17.563;
   1:L PR[91] R[100]mm/sec CNT100;
   1:  PR[GP1:91,1] = PR[GP1:90,1] + -19.911;
   1:  PR[GP1:91,2] = PR[GP1:90,2] + 18.212;
   1:L PR[91] R[100]mm/sec CNT100;
   1:  PR[GP1:91,1] = PR[GP1:90,1] + -21.781;
   1:  PR[GP1:91,2] = PR[GP1:90,2] + 18.491;
   1:L PR[91] R[100]mm/sec CNT100;
   1:  PR[GP1:91,1] = PR[GP1:90,1] + -23.928;
   1:  PR[GP1:91,2] = PR[GP1:90,2] + 18.292;
   1:L PR[91] R[100]mm/sec CNT100;
   1:  PR[GP1:91,1] = PR[GP1:90,1] + -26.046;
   1:  PR[GP1:91,2] = PR[GP1:90,2] + 18.259;
   1:L PR[91] R[100]mm/sec CNT100;
   1:  PR[GP1:91,1] = PR[GP1:90,1] + -27.905;
   1:  PR[GP1:91,2] = PR[GP1:90,2] + 17.922;
   1:L PR[91] R[100]mm/sec CNT100;
   1:  PR[GP1:91,1] = PR[GP1:90,1] + -29.873;
   1:  PR[GP1:91,2] = PR[GP1:90,2] + 17.041;
   1:L PR[91] R[100]mm/sec CNT100;
   1:  PR[GP1:91,1] = PR[GP1:90,1] + -31.869;
   1:  PR[GP1:91,2] = PR[GP1:90,2] + 16.327;
   1:L PR[91] R[100]mm/sec CNT100;
   1:  PR[GP1:91,1] = PR[GP1:90,1] + -33.520;
   1:  PR[GP1:91,2] = PR[GP1:90,2] + 15.411;
   1:L PR[91] R[100]mm/sec CNT100;
   1:  PR[GP1:91,1] = PR[GP1:90,1] + -35.099;
   1:  PR[GP1:91,2] = PR[GP1:90,2] + 13.942;
   1:L PR[91] R[100]mm/sec CNT100;
   1:  PR[GP1:91,1] = PR[GP1:90,1] + -36.760;
   1:  PR[GP1:91,2] = PR[GP1:90,2] + 12.624;
   1:L PR[91] R[100]mm/sec CNT100;
   1:  PR[GP1:91,1] = PR[GP1:90,1] + -38.028;
   1:  PR[GP1:91,2] = PR[GP1:90,2] + 11.226;
   1:L PR[91] R[100]mm/sec CNT100;
   1:  PR[GP1:91,1] = PR[GP1:90,1] + -39.049;
   1:  PR[GP1:91,2] = PR[GP1:90,2] + 9.326;
   1:L PR[91] R[100]mm/sec CNT100;
   1:  PR[GP1:91,1] = PR[GP1:90,1] + -40.199;
   1:  PR[GP1:91,2] = PR[GP1:90,2] + 7.544;
   1:L PR[91] R[100]mm/sec CNT100;
   1:  PR[GP1:91,1] = PR[GP1:90,1] + -40.949;
   1:  PR[GP1:91,2] = PR[GP1:90,2] + 5.813;
   1:L PR[91] R[100]mm/sec CNT100;
   1:  PR[GP1:91,1] = PR[GP1:90,1] + -41.302;
   1:  PR[GP1:91,2] = PR[GP1:90,2] + 3.686;
   1:L PR[91] R[100]mm/sec CNT100;
   1:  PR[GP1:91,1] = PR[GP1:90,1] + -41.818;
   1:  PR[GP1:91,2] = PR[GP1:90,2] + 1.627;
   1:L PR[91] R[100]mm/sec CNT100;
   1:  PR[GP1:91,1] = PR[GP1:90,1] + -41.972;
   1:  PR[GP1:91,2] = PR[GP1:90,2] + -0.252;
   1:L PR[91] R[100]mm/sec CNT100;
   1:  PR[GP1:91,1] = PR[GP1:90,1] + -41.619;
   1:  PR[GP1:91,2] = PR[GP1:90,2] + -2.380;
   1:L PR[91] R[100]mm/sec CNT100;
   1:  PR[GP1:91,1] = PR[GP1:90,1] + -41.446;
   1:  PR[GP1:91,2] = PR[GP1:90,2] + -4.496;
   1:L PR[91] R[100]mm/sec CNT100;
   1:  PR[GP1:91,1] = PR[GP1:90,1] + -40.973;
   1:  PR[GP1:91,2] = PR[GP1:90,2] + -6.383;
   1:L PR[91] R[100]mm/sec CNT100;
   1:  PR[GP1:91,1] = PR[GP1:90,1] + -40.176;
   1:  PR[GP1:91,2] = PR[GP1:90,2] + -8.221;
   1:L PR[91] R[100]mm/sec CNT100;
   1:  PR[GP1:91,1] = PR[GP1:90,1] + -39.155;
   1:  PR[GP1:91,2] = PR[GP1:90,2] + -10.121;
   1:L PR[91] R[100]mm/sec CNT100;
   1:  PR[GP1:91,1] = PR[GP1:90,1] + -38.067;
   1:  PR[GP1:91,2] = PR[GP1:90,2] + -11.807;
   1:L PR[91] R[100]mm/sec CNT100;
   1:  PR[GP1:91,1] = PR[GP1:90,1] + -36.722;
   1:  PR[GP1:91,2] = PR[GP1:90,2] + -13.290;
   1:L PR[91] R[100]mm/sec CNT100;
   1:  PR[GP1:91,1] = PR[GP1:90,1] + -35.143;
   1:  PR[GP1:91,2] = PR[GP1:90,2] + -14.760;
   1:L PR[91] R[100]mm/sec CNT100;
   1:  PR[GP1:91,1] = PR[GP1:90,1] + -33.570;
   1:  PR[GP1:91,2] = PR[GP1:90,2] + -16.007;
   1:L PR[91] R[100]mm/sec CNT100;
   1:  PR[GP1:91,1] = PR[GP1:90,1] + -31.820;
   1:  PR[GP1:91,2] = PR[GP1:90,2] + -16.979;
   1:L PR[91] R[100]mm/sec CNT100;
   1:  PR[GP1:91,1] = PR[GP1:90,1] + -29.851;
   1:  PR[GP1:91,2] = PR[GP1:90,2] + -17.860;
   1:L PR[91] R[100]mm/sec CNT100;
   1:  PR[GP1:91,1] = PR[GP1:90,1] + -27.961;
   1:  PR[GP1:91,2] = PR[GP1:90,2] + -18.535;
   1:L PR[91] R[100]mm/sec CNT100;
   1:  PR[GP1:91,1] = PR[GP1:90,1] + -25.992;
   1:  PR[GP1:91,2] = PR[GP1:90,2] + -18.893;
   1:L PR[91] R[100]mm/sec CNT100;
   1:  PR[GP1:91,1] = PR[GP1:90,1] + -23.844;
   1:  PR[GP1:91,2] = PR[GP1:90,2] + -19.091;
   1:L PR[91] R[100]mm/sec CNT100;
   1:  PR[GP1:91,1] = PR[GP1:90,1] + -21.836;
   1:  PR[GP1:91,2] = PR[GP1:90,2] + -19.123;
   1:L PR[91] R[100]mm/sec CNT100;
   1:  PR[GP1:91,1] = PR[GP1:90,1] + -19.857;
   1:  PR[GP1:91,2] = PR[GP1:90,2] + -18.828;
   1:L PR[91] R[100]mm/sec CNT100;
   1:  PR[GP1:91,1] = PR[GP1:90,1] + -17.760;
   1:  PR[GP1:91,2] = PR[GP1:90,2] + -18.323;
   1:L PR[91] R[100]mm/sec CNT100;
   1:  PR[GP1:91,1] = PR[GP1:90,1] + -15.848;
   1:  PR[GP1:91,2] = PR[GP1:90,2] + -17.707;
   1:L PR[91] R[100]mm/sec CNT100;
   1:  PR[GP1:91,1] = PR[GP1:90,1] + -14.070;
   1:  PR[GP1:91,2] = PR[GP1:90,2] + -16.792;
   1:L PR[91] R[100]mm/sec CNT100;
   1:  PR[GP1:91,1] = PR[GP1:90,1] + -12.248;
   1:  PR[GP1:91,2] = PR[GP1:90,2] + -15.638;
   1:L PR[91] R[100]mm/sec CNT100;
   1:  PR[GP1:91,1] = PR[GP1:90,1] + -10.634;
   1:  PR[GP1:91,2] = PR[GP1:90,2] + -14.439;
   1:L PR[91] R[100]mm/sec CNT100;
   1:  PR[GP1:91,1] = PR[GP1:90,1] + -9.246;
   1:  PR[GP1:91,2] = PR[GP1:90,2] + -13.002;
   1:L PR[91] R[100]mm/sec CNT100;
   1:  PR[GP1:91,1] = PR[GP1:90,1] + -7.894;
   1:  PR[GP1:91,2] = PR[GP1:90,2] + -11.322;
   1:L PR[91] R[100]mm/sec CNT100;
   1:  PR[GP1:91,1] = PR[GP1:90,1] + -6.751;
   1:  PR[GP1:91,2] = PR[GP1:90,2] + -9.667;
   1:L PR[91] R[100]mm/sec CNT100;
   1:  PR[GP1:91,1] = PR[GP1:90,1] + -5.899;
   1:  PR[GP1:91,2] = PR[GP1:90,2] + -7.860;
   1:L PR[91] R[100]mm/sec CNT100;
   1:  PR[GP1:91,1] = PR[GP1:90,1] + -5.162;
   1:  PR[GP1:91,2] = PR[GP1:90,2] + -5.836;
   1:L PR[91] R[100]mm/sec CNT100;
   1:  PR[GP1:91,1] = PR[GP1:90,1] + -4.596;
   1:  PR[GP1:91,2] = PR[GP1:90,2] + -3.848;
   1:L PR[91] R[100]mm/sec CNT100;
   1:  PR[GP1:91,1] = PR[GP1:90,1] + -4.559;
   1:  PR[GP1:91,2] = PR[GP1:90,2] + -3.655;
   1:L PR[91] R[100]mm/sec CNT100;
   1:  PR[GP1:91,1] = PR[GP1:90,1] + -4.206;
   1:  PR[GP1:91,2] = PR[GP1:90,2] + -2.731;
   1:L PR[91] R[100]mm/sec CNT100;
   1:  PR[GP1:91,1] = PR[GP1:90,1] + -3.610;
   1:  PR[GP1:91,2] = PR[GP1:90,2] + -2.030;
   1:L PR[91] R[100]mm/sec CNT100;
   1:  PR[GP1:91,1] = PR[GP1:90,1] + -3.365;
   1:  PR[GP1:91,2] = PR[GP1:90,2] + -1.826;
   1:L PR[91] R[100]mm/sec CNT100;
   1:  PR[GP1:91,1] = PR[GP1:90,1] + -2.566;
   1:  PR[GP1:91,2] = PR[GP1:90,2] + -1.370;
   1:L PR[91] R[100]mm/sec CNT100;
   1:  PR[GP1:91,1] = PR[GP1:90,1] + -1.589;
   1:  PR[GP1:91,2] = PR[GP1:90,2] + -1.192;
   1:L PR[91] R[100]mm/sec CNT100;
   1:  PR[GP1:91,1] = PR[GP1:90,1] + 1.745;
   1:L PR[91] R[100]mm/sec CNT100;
   1:  PR[GP1:91,1] = PR[GP1:90,1] + 2.723;
   1:  PR[GP1:91,2] = PR[GP1:90,2] + -1.370;
   1:L PR[91] R[100]mm/sec CNT100;
   1:  PR[GP1:91,1] = PR[GP1:90,1] + 3.522;
   1:  PR[GP1:91,2] = PR[GP1:90,2] + -1.826;
   1:L PR[91] R[100]mm/sec CNT100;
   1:  PR[GP1:91,1] = PR[GP1:90,1] + 3.767;
   1:  PR[GP1:91,2] = PR[GP1:90,2] + -2.030;
   1:L PR[91] R[100]mm/sec CNT100;
   1:  PR[GP1:91,1] = PR[GP1:90,1] + 4.366;
   1:  PR[GP1:91,2] = PR[GP1:90,2] + -2.735;
   1:L PR[91] R[100]mm/sec CNT100;
   1:  PR[GP1:91,1] = PR[GP1:90,1] + 4.875;
   1:  PR[GP1:91,2] = PR[GP1:90,2] + -4.098;
   1:L PR[91] R[100]mm/sec CNT100;
   1:  PR[GP1:91,1] = PR[GP1:90,1] + 5.502;
   1:  PR[GP1:91,2] = PR[GP1:90,2] + -5.880;
   1:L PR[91] R[100]mm/sec CNT100;
   1:  PR[GP1:91,1] = PR[GP1:90,1] + 6.078;
   1:  PR[GP1:91,2] = PR[GP1:90,2] + -7.907;
   1:L PR[91] R[100]mm/sec CNT100;
   1:  PR[GP1:91,1] = PR[GP1:90,1] + 6.885;
   1:  PR[GP1:91,2] = PR[GP1:90,2] + -9.619;
   1:L PR[91] R[100]mm/sec CNT100;
   1:  PR[GP1:91,1] = PR[GP1:90,1] + 8.237;
   1:  PR[GP1:91,2] = PR[GP1:90,2] + -11.299;
   1:L PR[91] R[100]mm/sec CNT100;
   1:  PR[GP1:91,1] = PR[GP1:90,1] + 9.440;
   1:  PR[GP1:91,2] = PR[GP1:90,2] + -13.040;
   1:L PR[91] R[100]mm/sec CNT100;
   1:  PR[GP1:91,1] = PR[GP1:90,1] + 10.754;
   1:  PR[GP1:91,2] = PR[GP1:90,2] + -14.400;
   1:L PR[91] R[100]mm/sec CNT100;
   1:  PR[GP1:91,1] = PR[GP1:90,1] + 12.575;
   1:  PR[GP1:91,2] = PR[GP1:90,2] + -15.554;
   1:L PR[91] R[100]mm/sec CNT100;
   1:  PR[GP1:91,1] = PR[GP1:90,1] + 14.275;
   1:  PR[GP1:91,2] = PR[GP1:90,2] + -16.817;
   1:L PR[91] R[100]mm/sec CNT100;
   1:  PR[GP1:91,1] = PR[GP1:90,1] + 15.956;
   1:  PR[GP1:91,2] = PR[GP1:90,2] + -17.682;
   1:L PR[91] R[100]mm/sec CNT100;
   1:  PR[GP1:91,1] = PR[GP1:90,1] + 18.052;
   1:  PR[GP1:91,2] = PR[GP1:90,2] + -18.187;
   1:L PR[91] R[100]mm/sec CNT100;
   1:  PR[GP1:91,1] = PR[GP1:90,1] + 20.068;
   1:  PR[GP1:91,2] = PR[GP1:90,2] + -18.836;
   1:L PR[91] R[100]mm/sec CNT100;
   1:  PR[GP1:91,1] = PR[GP1:90,1] + 21.937;
   1:  PR[GP1:91,2] = PR[GP1:90,2] + -19.115;
   1:L PR[91] R[100]mm/sec CNT100;
   1:  PR[GP1:91,1] = PR[GP1:90,1] + 24.085;
   1:  PR[GP1:91,2] = PR[GP1:90,2] + -18.916;
   1:L PR[91] R[100]mm/sec CNT100;
   1:  PR[GP1:91,1] = PR[GP1:90,1] + 26.203;
   1:  PR[GP1:91,2] = PR[GP1:90,2] + -18.883;
   1:L PR[91] R[100]mm/sec CNT100;
   1:  PR[GP1:91,1] = PR[GP1:90,1] + 28.062;
   1:  PR[GP1:91,2] = PR[GP1:90,2] + -18.546;
   1:L PR[91] R[100]mm/sec CNT100;
   1:  PR[GP1:91,1] = PR[GP1:90,1] + 30.030;
   1:  PR[GP1:91,2] = PR[GP1:90,2] + -17.665;
   1:L PR[91] R[100]mm/sec CNT100;
   1:  PR[GP1:91,1] = PR[GP1:90,1] + 32.026;
   1:  PR[GP1:91,2] = PR[GP1:90,2] + -16.951;
   1:L PR[91] R[100]mm/sec CNT100;
   1:  PR[GP1:91,1] = PR[GP1:90,1] + 33.677;
   1:  PR[GP1:91,2] = PR[GP1:90,2] + -16.035;
   1:L PR[91] R[100]mm/sec CNT100;
   1:  PR[GP1:91,1] = PR[GP1:90,1] + 35.256;
   1:  PR[GP1:91,2] = PR[GP1:90,2] + -14.566;
   1:L PR[91] R[100]mm/sec CNT100;
   1:  PR[GP1:91,1] = PR[GP1:90,1] + 36.917;
   1:  PR[GP1:91,2] = PR[GP1:90,2] + -13.248;
   1:L PR[91] R[100]mm/sec CNT100;
   1:  PR[GP1:91,1] = PR[GP1:90,1] + 38.185;
   1:  PR[GP1:91,2] = PR[GP1:90,2] + -11.850;
   1:L PR[91] R[100]mm/sec CNT100;
   1:  PR[GP1:91,1] = PR[GP1:90,1] + 39.205;
   1:  PR[GP1:91,2] = PR[GP1:90,2] + -9.950;
   1:L PR[91] R[100]mm/sec CNT100;
   1:  PR[GP1:91,1] = PR[GP1:90,1] + 40.355;
   1:  PR[GP1:91,2] = PR[GP1:90,2] + -8.168;
   1:L PR[91] R[100]mm/sec CNT100;
   1:  PR[GP1:91,1] = PR[GP1:90,1] + 41.106;
   1:  PR[GP1:91,2] = PR[GP1:90,2] + -6.437;
   1:L PR[91] R[100]mm/sec CNT100;
   1:  PR[GP1:91,1] = PR[GP1:90,1] + 41.459;
   1:  PR[GP1:91,2] = PR[GP1:90,2] + -4.310;
   1:L PR[91] R[100]mm/sec CNT100;
   1:  PR[GP1:91,1] = PR[GP1:90,1] + 41.974;
   1:  PR[GP1:91,2] = PR[GP1:90,2] + -2.251;
   1:L PR[91] R[100]mm/sec CNT100;
   1:  PR[GP1:91,1] = PR[GP1:90,1] + 42.129;
   1:  PR[GP1:91,2] = PR[GP1:90,2] + -0.372;
   1:L PR[91] R[100]mm/sec CNT100;
   1:  PR[GP1:91,1] = PR[GP1:90,1] + 41.776;
   1:  PR[GP1:91,2] = PR[GP1:90,2] + 1.756;
   1:L PR[91] R[100]mm/sec CNT100;
   1:  PR[GP1:91,1] = PR[GP1:90,1] + 41.602;
   1:  PR[GP1:91,2] = PR[GP1:90,2] + 3.872;
   1:L PR[91] R[100]mm/sec CNT100;
   1:  PR[GP1:91,1] = PR[GP1:90,1] + 41.129;
   1:  PR[GP1:91,2] = PR[GP1:90,2] + 5.759;
   1:L PR[91] R[100]mm/sec CNT100;
   1:  PR[GP1:91,1] = PR[GP1:90,1] + 40.332;
   1:  PR[GP1:91,2] = PR[GP1:90,2] + 7.597;
   1:L PR[91] R[100]mm/sec CNT100;
   1:  PR[GP1:91,1] = PR[GP1:90,1] + 39.312;
   1:  PR[GP1:91,2] = PR[GP1:90,2] + 9.497;
   1:L PR[91] R[100]mm/sec CNT100;
   1:  PR[GP1:91,1] = PR[GP1:90,1] + 38.224;
   1:  PR[GP1:91,2] = PR[GP1:90,2] + 11.183;
   1:L PR[91] R[100]mm/sec CNT100;
   1:  PR[GP1:91,1] = PR[GP1:90,1] + 36.879;
   1:  PR[GP1:91,2] = PR[GP1:90,2] + 12.666;
   1:L PR[91] R[100]mm/sec CNT100;
   1:  PR[GP1:91,1] = PR[GP1:90,1] + 35.300;
   1:  PR[GP1:91,2] = PR[GP1:90,2] + 14.136;
   1:L PR[91] R[100]mm/sec CNT100;
   1:  PR[GP1:91,1] = PR[GP1:90,1] + 33.727;
   1:  PR[GP1:91,2] = PR[GP1:90,2] + 15.383;
   1:L PR[91] R[100]mm/sec CNT100;
   1:  PR[GP1:91,1] = PR[GP1:90,1] + 31.977;
   1:  PR[GP1:91,2] = PR[GP1:90,2] + 16.355;
   1:L PR[91] R[100]mm/sec CNT100;
   1:  PR[GP1:91,1] = PR[GP1:90,1] + 30.008;
   1:  PR[GP1:91,2] = PR[GP1:90,2] + 17.236;
   1:L PR[91] R[100]mm/sec CNT100;
   1:  PR[GP1:91,1] = PR[GP1:90,1] + 28.117;
   1:  PR[GP1:91,2] = PR[GP1:90,2] + 17.911;
   1:L PR[91] R[100]mm/sec CNT100;
   1:  PR[GP1:91,1] = PR[GP1:90,1] + 26.149;
   1:  PR[GP1:91,2] = PR[GP1:90,2] + 18.269;
   1:L PR[91] R[100]mm/sec CNT100;
   1:  PR[GP1:91,1] = PR[GP1:90,1] + 24.001;
   1:  PR[GP1:91,2] = PR[GP1:90,2] + 18.467;
   1:L PR[91] R[100]mm/sec CNT100;
   1:  PR[GP1:91,1] = PR[GP1:90,1] + 21.992;
   1:  PR[GP1:91,2] = PR[GP1:90,2] + 18.499;
   1:L PR[91] R[100]mm/sec CNT100;
   1:  PR[GP1:91,1] = PR[GP1:90,1] + 20.014;
   1:  PR[GP1:91,2] = PR[GP1:90,2] + 18.204;
   1:L PR[91] R[100]mm/sec CNT100;
   1:  PR[GP1:91,1] = PR[GP1:90,1] + 17.917;
   1:  PR[GP1:91,2] = PR[GP1:90,2] + 17.699;
   1:L PR[91] R[100]mm/sec CNT100;
   1:  PR[GP1:91,1] = PR[GP1:90,1] + 16.004;
   1:  PR[GP1:91,2] = PR[GP1:90,2] + 17.083;
   1:L PR[91] R[100]mm/sec CNT100;
   1:  PR[GP1:91,1] = PR[GP1:90,1] + 14.227;
   1:  PR[GP1:91,2] = PR[GP1:90,2] + 16.169;
   1:L PR[91] R[100]mm/sec CNT100;
   1:  PR[GP1:91,1] = PR[GP1:90,1] + 12.405;
   1:  PR[GP1:91,2] = PR[GP1:90,2] + 15.014;
   1:L PR[91] R[100]mm/sec CNT100;
   1:  PR[GP1:91,1] = PR[GP1:90,1] + 10.791;
   1:  PR[GP1:91,2] = PR[GP1:90,2] + 13.815;
   1:L PR[91] R[100]mm/sec CNT100;
   1:  PR[GP1:91,1] = PR[GP1:90,1] + 9.403;
   1:  PR[GP1:91,2] = PR[GP1:90,2] + 12.378;
   1:L PR[91] R[100]mm/sec CNT100;
   1:  PR[GP1:91,1] = PR[GP1:90,1] + 8.051;
   1:  PR[GP1:91,2] = PR[GP1:90,2] + 10.698;
   1:L PR[91] R[100]mm/sec CNT100;
   1:  PR[GP1:91,1] = PR[GP1:90,1] + 6.908;
   1:  PR[GP1:91,2] = PR[GP1:90,2] + 9.043;
   1:L PR[91] R[100]mm/sec CNT100;
   1:  PR[GP1:91,1] = PR[GP1:90,1] + 6.056;
   1:  PR[GP1:91,2] = PR[GP1:90,2] + 7.236;
   1:L PR[91] R[100]mm/sec CNT100;
   1:  PR[GP1:91,1] = PR[GP1:90,1] + 5.318;
   1:  PR[GP1:91,2] = PR[GP1:90,2] + 5.212;
   1:L PR[91] R[100]mm/sec CNT100;
   1:  PR[GP1:91,1] = PR[GP1:90,1] + 4.753;
   1:  PR[GP1:91,2] = PR[GP1:90,2] + 3.224;
   1:L PR[91] R[100]mm/sec CNT100;
   1:  PR[GP1:91,1] = PR[GP1:90,1] + 4.716;
   1:  PR[GP1:91,2] = PR[GP1:90,2] + 3.031;
   1:L PR[91] R[100]mm/sec CNT100;
   1:  PR[GP1:91,1] = PR[GP1:90,1] + 4.363;
   1:  PR[GP1:91,2] = PR[GP1:90,2] + 2.107;
   1:L PR[91] R[100]mm/sec CNT100;
   1:  PR[GP1:91,1] = PR[GP1:90,1] + 3.767;
   1:  PR[GP1:91,2] = PR[GP1:90,2] + 1.406;
   1:L PR[91] R[100]mm/sec CNT100;
   1:  PR[GP1:91,1] = PR[GP1:90,1] + 3.522;
   1:  PR[GP1:91,2] = PR[GP1:90,2] + 1.202;
   1:L PR[91] R[100]mm/sec CNT100;
   1:  PR[GP1:91,1] = PR[GP1:90,1] + 2.723;
   1:  PR[GP1:91,2] = PR[GP1:90,2] + 0.746;
   1:L PR[91] R[100]mm/sec CNT100;
   1:  PR[GP1:91,1] = PR[GP1:90,1] + 1.745;
   1:  PR[GP1:91,2] = PR[GP1:90,2] + 0.568;
   1:L PR[91] R[100]mm/sec CNT100;
   1:  PR[GP1:91,1] = PR[GP1:90,1] + -1.589;
   1:L PR[91] R[100]mm/sec CNT100;
   1:  PR[91] = PR[90];
   1:  PR[GP1:91,1] = PR[GP1:90,1] + -1.983;
   1:  PR[GP1:91,2] = PR[GP1:90,2] + 0.688;
   1:  PR[GP1:91,3] = PR[GP1:90,3] + 3.965;
   1:L PR[91] R[100]mm/sec CNT100;
   1:  PR[GP1:91,1] = PR[GP1:90,1] + -2.552;
   1:  PR[GP1:91,2] = PR[GP1:90,2] + 0.788;
   1:L PR[91] R[100]mm/sec CNT100;
   1:  PR[GP1:91,1] = PR[GP1:90,1] + -3.509;
   1:  PR[GP1:91,2] = PR[GP1:90,2] + 1.333;
   1:L PR[91] R[100]mm/sec CNT100;
   1:  PR[GP1:91,1] = PR[GP1:90,1] + -4.222;
   1:  PR[GP1:91,2] = PR[GP1:90,2] + 2.167;
   1:L PR[91] R[100]mm/sec CNT100;
   1:  PR[GP1:91,1] = PR[GP1:90,1] + -4.525;
   1:  PR[GP1:91,2] = PR[GP1:90,2] + 2.953;
   1:L PR[91] R[100]mm/sec CNT100;
   1:  PR[GP1:91,1] = PR[GP1:90,1] + -5.052;
   1:  PR[GP1:91,2] = PR[GP1:90,2] + 4.465;
   1:L PR[91] R[100]mm/sec CNT100;
   1:  PR[GP1:91,1] = PR[GP1:90,1] + -5.747;
   1:  PR[GP1:91,2] = PR[GP1:90,2] + 6.910;
   1:L PR[91] R[100]mm/sec CNT100;
   1:  PR[GP1:91,1] = PR[GP1:90,1] + -6.741;
   1:  PR[GP1:91,2] = PR[GP1:90,2] + 9.016;
   1:L PR[91] R[100]mm/sec CNT100;
   1:  PR[GP1:91,1] = PR[GP1:90,1] + -7.545;
   1:  PR[GP1:91,2] = PR[GP1:90,2] + 10.016;
   1:L PR[91] R[100]mm/sec CNT100;
   1:  PR[GP1:91,1] = PR[GP1:90,1] + -8.996;
   1:  PR[GP1:91,2] = PR[GP1:90,2] + 12.117;
   1:L PR[91] R[100]mm/sec CNT100;
   1:  PR[GP1:91,1] = PR[GP1:90,1] + -10.613;
   1:  PR[GP1:91,2] = PR[GP1:90,2] + 13.791;
   1:L PR[91] R[100]mm/sec CNT100;
   1:  PR[GP1:91,1] = PR[GP1:90,1] + -11.697;
   1:  PR[GP1:91,2] = PR[GP1:90,2] + 14.478;
   1:L PR[91] R[100]mm/sec CNT100;
   1:  PR[GP1:91,1] = PR[GP1:90,1] + -13.747;
   1:  PR[GP1:91,2] = PR[GP1:90,2] + 16.001;
   1:L PR[91] R[100]mm/sec CNT100;
   1:  PR[GP1:91,1] = PR[GP1:90,1] + -15.816;
   1:  PR[GP1:91,2] = PR[GP1:90,2] + 17.066;
   1:L PR[91] R[100]mm/sec CNT100;
   1:  PR[GP1:91,1] = PR[GP1:90,1] + -17.064;
   1:  PR[GP1:91,2] = PR[GP1:90,2] + 17.366;
   1:L PR[91] R[100]mm/sec CNT100;
   1:  PR[GP1:91,1] = PR[GP1:90,1] + -19.495;
   1:  PR[GP1:91,2] = PR[GP1:90,2] + 18.149;
   1:L PR[91] R[100]mm/sec CNT100;
   1:  PR[GP1:91,1] = PR[GP1:90,1] + -21.796;
   1:  PR[GP1:91,2] = PR[GP1:90,2] + 18.492;
   1:L PR[91] R[100]mm/sec CNT100;
   1:  PR[GP1:91,1] = PR[GP1:90,1] + -23.074;
   1:  PR[GP1:91,2] = PR[GP1:90,2] + 18.374;
   1:L PR[91] R[100]mm/sec CNT100;
   1:  PR[GP1:91,1] = PR[GP1:90,1] + -25.629;
   1:  PR[GP1:91,2] = PR[GP1:90,2] + 18.333;
   1:L PR[91] R[100]mm/sec CNT100;
   1:  PR[GP1:91,1] = PR[GP1:90,1] + -27.917;
   1:  PR[GP1:91,2] = PR[GP1:90,2] + 17.918;
   1:L PR[91] R[100]mm/sec CNT100;
   1:  PR[GP1:91,1] = PR[GP1:90,1] + -29.089;
   1:  PR[GP1:91,2] = PR[GP1:90,2] + 17.394;
   1:L PR[91] R[100]mm/sec CNT100;
   1:  PR[GP1:91,1] = PR[GP1:90,1] + -31.496;
   1:  PR[GP1:91,2] = PR[GP1:90,2] + 16.534;
   1:L PR[91] R[100]mm/sec CNT100;
   1:  PR[GP1:91,1] = PR[GP1:90,1] + -33.528;
   1:  PR[GP1:91,2] = PR[GP1:90,2] + 15.406;
   1:L PR[91] R[100]mm/sec CNT100;
   1:  PR[GP1:91,1] = PR[GP1:90,1] + -34.468;
   1:  PR[GP1:91,2] = PR[GP1:90,2] + 14.531;
   1:L PR[91] R[100]mm/sec CNT100;
   1:  PR[GP1:91,1] = PR[GP1:90,1] + -36.471;
   1:  PR[GP1:91,2] = PR[GP1:90,2] + 12.943;
   1:L PR[91] R[100]mm/sec CNT100;
   1:  PR[GP1:91,1] = PR[GP1:90,1] + -38.032;
   1:  PR[GP1:91,2] = PR[GP1:90,2] + 11.221;
   1:L PR[91] R[100]mm/sec CNT100;
   1:  PR[GP1:91,1] = PR[GP1:90,1] + -38.639;
   1:  PR[GP1:91,2] = PR[GP1:90,2] + 10.090;
   1:L PR[91] R[100]mm/sec CNT100;
   1:  PR[GP1:91,1] = PR[GP1:90,1] + -40.026;
   1:  PR[GP1:91,2] = PR[GP1:90,2] + 7.941;
   1:L PR[91] R[100]mm/sec CNT100;
   1:  PR[GP1:91,1] = PR[GP1:90,1] + -40.950;
   1:  PR[GP1:91,2] = PR[GP1:90,2] + 5.810;
   1:L PR[91] R[100]mm/sec CNT100;
   1:  PR[GP1:91,1] = PR[GP1:90,1] + -41.160;
   1:  PR[GP1:91,2] = PR[GP1:90,2] + 4.544;
   1:L PR[91] R[100]mm/sec CNT100;
   1:  PR[GP1:91,1] = PR[GP1:90,1] + -41.782;
   1:  PR[GP1:91,2] = PR[GP1:90,2] + 2.062;
   1:L PR[91] R[100]mm/sec CNT100;
   1:  PR[GP1:91,1] = PR[GP1:90,1] + -41.972;
   1:  PR[GP1:91,2] = PR[GP1:90,2] + -0.252;
   1:L PR[91] R[100]mm/sec CNT100;
   1:  PR[GP1:91,1] = PR[GP1:90,1] + -41.762;
   1:  PR[GP1:91,2] = PR[GP1:90,2] + -1.519;
   1:L PR[91] R[100]mm/sec CNT100;
   1:  PR[GP1:91,1] = PR[GP1:90,1] + -41.553;
   1:  PR[GP1:91,2] = PR[GP1:90,2] + -4.069;
   1:L PR[91] R[100]mm/sec CNT100;
   1:  PR[GP1:91,1] = PR[GP1:90,1] + -40.974;
   1:  PR[GP1:91,2] = PR[GP1:90,2] + -6.380;
   1:L PR[91] R[100]mm/sec CNT100;
   1:  PR[GP1:91,1] = PR[GP1:90,1] + -40.003;
   1:  PR[GP1:91,2] = PR[GP1:90,2] + -8.618;
   1:L PR[91] R[100]mm/sec CNT100;
   1:  PR[GP1:91,1] = PR[GP1:90,1] + -39.395;
   1:  PR[GP1:91,2] = PR[GP1:90,2] + -9.750;
   1:L PR[91] R[100]mm/sec CNT100;
   1:  PR[GP1:91,1] = PR[GP1:90,1] + -38.071;
   1:  PR[GP1:91,2] = PR[GP1:90,2] + -11.802;
   1:L PR[91] R[100]mm/sec CNT100;
   1:  PR[GP1:91,1] = PR[GP1:90,1] + -36.433;
   1:  PR[GP1:91,2] = PR[GP1:90,2] + -13.609;
   1:L PR[91] R[100]mm/sec CNT100;
   1:  PR[GP1:91,1] = PR[GP1:90,1] + -35.492;
   1:  PR[GP1:91,2] = PR[GP1:90,2] + -14.484;
   1:L PR[91] R[100]mm/sec CNT100;
   1:  PR[GP1:91,1] = PR[GP1:90,1] + -33.578;
   1:  PR[GP1:91,2] = PR[GP1:90,2] + -16.002;
   1:L PR[91] R[100]mm/sec CNT100;
   1:  PR[GP1:91,1] = PR[GP1:90,1] + -31.447;
   1:  PR[GP1:91,2] = PR[GP1:90,2] + -17.185;
   1:L PR[91] R[100]mm/sec CNT100;
   1:  PR[GP1:91,1] = PR[GP1:90,1] + -30.274;
   1:  PR[GP1:91,2] = PR[GP1:90,2] + -17.710;
   1:L PR[91] R[100]mm/sec CNT100;
   1:  PR[GP1:91,1] = PR[GP1:90,1] + -27.973;
   1:  PR[GP1:91,2] = PR[GP1:90,2] + -18.532;
   1:L PR[91] R[100]mm/sec CNT100;
   1:  PR[GP1:91,1] = PR[GP1:90,1] + -25.575;
   1:  PR[GP1:91,2] = PR[GP1:90,2] + -18.967;
   1:L PR[91] R[100]mm/sec CNT100;
   1:  PR[GP1:91,1] = PR[GP1:90,1] + -24.296;
   1:  PR[GP1:91,2] = PR[GP1:90,2] + -19.086;
   1:L PR[91] R[100]mm/sec CNT100;
   1:  PR[GP1:91,1] = PR[GP1:90,1] + -21.851;
   1:  PR[GP1:91,2] = PR[GP1:90,2] + -19.124;
   1:L PR[91] R[100]mm/sec CNT100;
   1:  PR[GP1:91,1] = PR[GP1:90,1] + -19.441;
   1:  PR[GP1:91,2] = PR[GP1:90,2] + -18.765;
   1:L PR[91] R[100]mm/sec CNT100;
   1:  PR[GP1:91,1] = PR[GP1:90,1] + -18.193;
   1:  PR[GP1:91,2] = PR[GP1:90,2] + -18.465;
   1:L PR[91] R[100]mm/sec CNT100;
   1:  PR[GP1:91,1] = PR[GP1:90,1] + -15.865;
   1:  PR[GP1:91,2] = PR[GP1:90,2] + -17.715;
   1:L PR[91] R[100]mm/sec CNT100;
   1:  PR[GP1:91,1] = PR[GP1:90,1] + -13.699;
   1:  PR[GP1:91,2] = PR[GP1:90,2] + -16.600;
   1:L PR[91] R[100]mm/sec CNT100;
   1:  PR[GP1:91,1] = PR[GP1:90,1] + -12.614;
   1:  PR[GP1:91,2] = PR[GP1:90,2] + -15.913;
   1:L PR[91] R[100]mm/sec CNT100;
   1:  PR[GP1:91,1] = PR[GP1:90,1] + -10.651;
   1:  PR[GP1:91,2] = PR[GP1:90,2] + -14.454;
   1:L PR[91] R[100]mm/sec CNT100;
   1:  PR[GP1:91,1] = PR[GP1:90,1] + -8.959;
   1:  PR[GP1:91,2] = PR[GP1:90,2] + -12.702;
   1:L PR[91] R[100]mm/sec CNT100;
   1:  PR[GP1:91,1] = PR[GP1:90,1] + -8.154;
   1:  PR[GP1:91,2] = PR[GP1:90,2] + -11.702;
   1:L PR[91] R[100]mm/sec CNT100;
   1:  PR[GP1:91,1] = PR[GP1:90,1] + -6.763;
   1:  PR[GP1:91,2] = PR[GP1:90,2] + -9.688;
   1:L PR[91] R[100]mm/sec CNT100;
   1:  PR[GP1:91,1] = PR[GP1:90,1] + -5.725;
   1:  PR[GP1:91,2] = PR[GP1:90,2] + -7.487;
   1:L PR[91] R[100]mm/sec CNT100;
   1:  PR[GP1:91,1] = PR[GP1:90,1] + -5.286;
   1:  PR[GP1:91,2] = PR[GP1:90,2] + -6.282;
   1:L PR[91] R[100]mm/sec CNT100;
   1:  PR[GP1:91,1] = PR[GP1:90,1] + -4.601;
   1:  PR[GP1:91,2] = PR[GP1:90,2] + -3.873;
   1:L PR[91] R[100]mm/sec CNT100;
   1:  PR[GP1:91,1] = PR[GP1:90,1] + -4.563;
   1:  PR[GP1:91,2] = PR[GP1:90,2] + -3.677;
   1:L PR[91] R[100]mm/sec CNT100;
   1:  PR[GP1:91,1] = PR[GP1:90,1] + -4.222;
   1:  PR[GP1:91,2] = PR[GP1:90,2] + -2.792;
   1:L PR[91] R[100]mm/sec CNT100;
   1:  PR[GP1:91,1] = PR[GP1:90,1] + -3.509;
   1:  PR[GP1:91,2] = PR[GP1:90,2] + -1.957;
   1:L PR[91] R[100]mm/sec CNT100;
   1:  PR[GP1:91,1] = PR[GP1:90,1] + -2.552;
   1:  PR[GP1:91,2] = PR[GP1:90,2] + -1.412;
   1:L PR[91] R[100]mm/sec CNT100;
   1:  PR[GP1:91,1] = PR[GP1:90,1] + -1.968;
   1:  PR[GP1:91,2] = PR[GP1:90,2] + -1.310;
   1:L PR[91] R[100]mm/sec CNT100;
   1:  PR[GP1:91,1] = PR[GP1:90,1] + -1.740;
   1:  PR[GP1:91,2] = PR[GP1:90,2] + -1.219;
   1:L PR[91] R[100]mm/sec CNT100;
   1:  PR[GP1:91,1] = PR[GP1:90,1] + 1.911;
   1:  PR[GP1:91,2] = PR[GP1:90,2] + -1.216;
   1:L PR[91] R[100]mm/sec CNT100;
   1:  PR[GP1:91,1] = PR[GP1:90,1] + 2.139;
   1:  PR[GP1:91,2] = PR[GP1:90,2] + -1.313;
   1:L PR[91] R[100]mm/sec CNT100;
   1:  PR[GP1:91,1] = PR[GP1:90,1] + 2.708;
   1:  PR[GP1:91,2] = PR[GP1:90,2] + -1.412;
   1:L PR[91] R[100]mm/sec CNT100;
   1:  PR[GP1:91,1] = PR[GP1:90,1] + 3.666;
   1:  PR[GP1:91,2] = PR[GP1:90,2] + -1.957;
   1:L PR[91] R[100]mm/sec CNT100;
   1:  PR[GP1:91,1] = PR[GP1:90,1] + 4.378;
   1:  PR[GP1:91,2] = PR[GP1:90,2] + -2.791;
   1:L PR[91] R[100]mm/sec CNT100;
   1:  PR[GP1:91,1] = PR[GP1:90,1] + 4.682;
   1:  PR[GP1:91,2] = PR[GP1:90,2] + -3.577;
   1:L PR[91] R[100]mm/sec CNT100;
   1:  PR[GP1:91,1] = PR[GP1:90,1] + 5.209;
   1:  PR[GP1:91,2] = PR[GP1:90,2] + -5.089;
   1:L PR[91] R[100]mm/sec CNT100;
   1:  PR[GP1:91,1] = PR[GP1:90,1] + 5.904;
   1:  PR[GP1:91,2] = PR[GP1:90,2] + -7.534;
   1:L PR[91] R[100]mm/sec CNT100;
   1:  PR[GP1:91,1] = PR[GP1:90,1] + 6.897;
   1:  PR[GP1:91,2] = PR[GP1:90,2] + -9.640;
   1:L PR[91] R[100]mm/sec CNT100;
   1:  PR[GP1:91,1] = PR[GP1:90,1] + 7.702;
   1:  PR[GP1:91,2] = PR[GP1:90,2] + -10.640;
   1:L PR[91] R[100]mm/sec CNT100;
   1:  PR[GP1:91,1] = PR[GP1:90,1] + 9.153;
   1:  PR[GP1:91,2] = PR[GP1:90,2] + -12.741;
   1:L PR[91] R[100]mm/sec CNT100;
   1:  PR[GP1:91,1] = PR[GP1:90,1] + 10.770;
   1:  PR[GP1:91,2] = PR[GP1:90,2] + -14.415;
   1:L PR[91] R[100]mm/sec CNT100;
   1:  PR[GP1:91,1] = PR[GP1:90,1] + 11.854;
   1:  PR[GP1:91,2] = PR[GP1:90,2] + -15.102;
   1:L PR[91] R[100]mm/sec CNT100;
   1:  PR[GP1:91,1] = PR[GP1:90,1] + 13.904;
   1:  PR[GP1:91,2] = PR[GP1:90,2] + -16.625;
   1:L PR[91] R[100]mm/sec CNT100;
   1:  PR[GP1:91,1] = PR[GP1:90,1] + 15.973;
   1:  PR[GP1:91,2] = PR[GP1:90,2] + -17.690;
   1:L PR[91] R[100]mm/sec CNT100;
   1:  PR[GP1:91,1] = PR[GP1:90,1] + 17.221;
   1:  PR[GP1:91,2] = PR[GP1:90,2] + -17.990;
   1:L PR[91] R[100]mm/sec CNT100;
   1:  PR[GP1:91,1] = PR[GP1:90,1] + 19.652;
   1:  PR[GP1:91,2] = PR[GP1:90,2] + -18.773;
   1:L PR[91] R[100]mm/sec CNT100;
   1:  PR[GP1:91,1] = PR[GP1:90,1] + 21.953;
   1:  PR[GP1:91,2] = PR[GP1:90,2] + -19.116;
   1:L PR[91] R[100]mm/sec CNT100;
   1:  PR[GP1:91,1] = PR[GP1:90,1] + 23.231;
   1:  PR[GP1:91,2] = PR[GP1:90,2] + -18.998;
   1:L PR[91] R[100]mm/sec CNT100;
   1:  PR[GP1:91,1] = PR[GP1:90,1] + 25.786;
   1:  PR[GP1:91,2] = PR[GP1:90,2] + -18.957;
   1:L PR[91] R[100]mm/sec CNT100;
   1:  PR[GP1:91,1] = PR[GP1:90,1] + 28.074;
   1:  PR[GP1:91,2] = PR[GP1:90,2] + -18.542;
   1:L PR[91] R[100]mm/sec CNT100;
   1:  PR[GP1:91,1] = PR[GP1:90,1] + 29.246;
   1:  PR[GP1:91,2] = PR[GP1:90,2] + -18.018;
   1:L PR[91] R[100]mm/sec CNT100;
   1:  PR[GP1:91,1] = PR[GP1:90,1] + 31.653;
   1:  PR[GP1:91,2] = PR[GP1:90,2] + -17.158;
   1:L PR[91] R[100]mm/sec CNT100;
   1:  PR[GP1:91,1] = PR[GP1:90,1] + 33.685;
   1:  PR[GP1:91,2] = PR[GP1:90,2] + -16.030;
   1:L PR[91] R[100]mm/sec CNT100;
   1:  PR[GP1:91,1] = PR[GP1:90,1] + 34.625;
   1:  PR[GP1:91,2] = PR[GP1:90,2] + -15.155;
   1:L PR[91] R[100]mm/sec CNT100;
   1:  PR[GP1:91,1] = PR[GP1:90,1] + 36.628;
   1:  PR[GP1:91,2] = PR[GP1:90,2] + -13.566;
   1:L PR[91] R[100]mm/sec CNT100;
   1:  PR[GP1:91,1] = PR[GP1:90,1] + 38.189;
   1:  PR[GP1:91,2] = PR[GP1:90,2] + -11.845;
   1:L PR[91] R[100]mm/sec CNT100;
   1:  PR[GP1:91,1] = PR[GP1:90,1] + 38.796;
   1:  PR[GP1:91,2] = PR[GP1:90,2] + -10.714;
   1:L PR[91] R[100]mm/sec CNT100;
   1:  PR[GP1:91,1] = PR[GP1:90,1] + 40.183;
   1:  PR[GP1:91,2] = PR[GP1:90,2] + -8.565;
   1:L PR[91] R[100]mm/sec CNT100;
   1:  PR[GP1:91,1] = PR[GP1:90,1] + 41.107;
   1:  PR[GP1:91,2] = PR[GP1:90,2] + -6.434;
   1:L PR[91] R[100]mm/sec CNT100;
   1:  PR[GP1:91,1] = PR[GP1:90,1] + 41.317;
   1:  PR[GP1:91,2] = PR[GP1:90,2] + -5.168;
   1:L PR[91] R[100]mm/sec CNT100;
   1:  PR[GP1:91,1] = PR[GP1:90,1] + 41.939;
   1:  PR[GP1:91,2] = PR[GP1:90,2] + -2.686;
   1:L PR[91] R[100]mm/sec CNT100;
   1:  PR[GP1:91,1] = PR[GP1:90,1] + 42.129;
   1:  PR[GP1:91,2] = PR[GP1:90,2] + -0.372;
   1:L PR[91] R[100]mm/sec CNT100;
   1:  PR[GP1:91,1] = PR[GP1:90,1] + 41.919;
   1:  PR[GP1:91,2] = PR[GP1:90,2] + 0.895;
   1:L PR[91] R[100]mm/sec CNT100;
   1:  PR[GP1:91,1] = PR[GP1:90,1] + 41.709;
   1:  PR[GP1:91,2] = PR[GP1:90,2] + 3.445;
   1:L PR[91] R[100]mm/sec CNT100;
   1:  PR[GP1:91,1] = PR[GP1:90,1] + 41.130;
   1:  PR[GP1:91,2] = PR[GP1:90,2] + 5.756;
   1:L PR[91] R[100]mm/sec CNT100;
   1:  PR[GP1:91,1] = PR[GP1:90,1] + 40.160;
   1:  PR[GP1:91,2] = PR[GP1:90,2] + 7.994;
   1:L PR[91] R[100]mm/sec CNT100;
   1:  PR[GP1:91,1] = PR[GP1:90,1] + 39.552;
   1:  PR[GP1:91,2] = PR[GP1:90,2] + 9.126;
   1:L PR[91] R[100]mm/sec CNT100;
   1:  PR[GP1:91,1] = PR[GP1:90,1] + 38.228;
   1:  PR[GP1:91,2] = PR[GP1:90,2] + 11.178;
   1:L PR[91] R[100]mm/sec CNT100;
   1:  PR[GP1:91,1] = PR[GP1:90,1] + 36.590;
   1:  PR[GP1:91,2] = PR[GP1:90,2] + 12.985;
   1:L PR[91] R[100]mm/sec CNT100;
   1:  PR[GP1:91,1] = PR[GP1:90,1] + 35.649;
   1:  PR[GP1:91,2] = PR[GP1:90,2] + 13.860;
   1:L PR[91] R[100]mm/sec CNT100;
   1:  PR[GP1:91,1] = PR[GP1:90,1] + 33.735;
   1:  PR[GP1:91,2] = PR[GP1:90,2] + 15.378;
   1:L PR[91] R[100]mm/sec CNT100;
   1:  PR[GP1:91,1] = PR[GP1:90,1] + 31.603;
   1:  PR[GP1:91,2] = PR[GP1:90,2] + 16.561;
   1:L PR[91] R[100]mm/sec CNT100;
   1:  PR[GP1:91,1] = PR[GP1:90,1] + 30.431;
   1:  PR[GP1:91,2] = PR[GP1:90,2] + 17.086;
   1:L PR[91] R[100]mm/sec CNT100;
   1:  PR[GP1:91,1] = PR[GP1:90,1] + 28.130;
   1:  PR[GP1:91,2] = PR[GP1:90,2] + 17.908;
   1:L PR[91] R[100]mm/sec CNT100;
   1:  PR[GP1:91,1] = PR[GP1:90,1] + 25.731;
   1:  PR[GP1:91,2] = PR[GP1:90,2] + 18.343;
   1:L PR[91] R[100]mm/sec CNT100;
   1:  PR[GP1:91,1] = PR[GP1:90,1] + 24.452;
   1:  PR[GP1:91,2] = PR[GP1:90,2] + 18.462;
   1:L PR[91] R[100]mm/sec CNT100;
   1:  PR[GP1:91,1] = PR[GP1:90,1] + 22.008;
   1:  PR[GP1:91,2] = PR[GP1:90,2] + 18.500;
   1:L PR[91] R[100]mm/sec CNT100;
   1:  PR[GP1:91,1] = PR[GP1:90,1] + 19.598;
   1:  PR[GP1:91,2] = PR[GP1:90,2] + 18.141;
   1:L PR[91] R[100]mm/sec CNT100;
   1:  PR[GP1:91,1] = PR[GP1:90,1] + 18.350;
   1:  PR[GP1:91,2] = PR[GP1:90,2] + 17.840;
   1:L PR[91] R[100]mm/sec CNT100;
   1:  PR[GP1:91,1] = PR[GP1:90,1] + 16.022;
   1:  PR[GP1:91,2] = PR[GP1:90,2] + 17.091;
   1:L PR[91] R[100]mm/sec CNT100;
   1:  PR[GP1:91,1] = PR[GP1:90,1] + 13.856;
   1:  PR[GP1:91,2] = PR[GP1:90,2] + 15.976;
   1:L PR[91] R[100]mm/sec CNT100;
   1:  PR[GP1:91,1] = PR[GP1:90,1] + 12.771;
   1:  PR[GP1:91,2] = PR[GP1:90,2] + 15.289;
   1:L PR[91] R[100]mm/sec CNT100;
   1:  PR[GP1:91,1] = PR[GP1:90,1] + 10.807;
   1:  PR[GP1:91,2] = PR[GP1:90,2] + 13.830;
   1:L PR[91] R[100]mm/sec CNT100;
   1:  PR[GP1:91,1] = PR[GP1:90,1] + 9.116;
   1:  PR[GP1:91,2] = PR[GP1:90,2] + 12.079;
   1:L PR[91] R[100]mm/sec CNT100;
   1:  PR[GP1:91,1] = PR[GP1:90,1] + 8.311;
   1:  PR[GP1:91,2] = PR[GP1:90,2] + 11.078;
   1:L PR[91] R[100]mm/sec CNT100;
   1:  PR[GP1:91,1] = PR[GP1:90,1] + 6.920;
   1:  PR[GP1:91,2] = PR[GP1:90,2] + 9.064;
   1:L PR[91] R[100]mm/sec CNT100;
   1:  PR[GP1:91,1] = PR[GP1:90,1] + 5.882;
   1:  PR[GP1:91,2] = PR[GP1:90,2] + 6.863;
   1:L PR[91] R[100]mm/sec CNT100;
   1:  PR[GP1:91,1] = PR[GP1:90,1] + 5.443;
   1:  PR[GP1:91,2] = PR[GP1:90,2] + 5.658;
   1:L PR[91] R[100]mm/sec CNT100;
   1:  PR[GP1:91,1] = PR[GP1:90,1] + 4.758;
   1:  PR[GP1:91,2] = PR[GP1:90,2] + 3.249;
   1:L PR[91] R[100]mm/sec CNT100;
   1:  PR[GP1:91,1] = PR[GP1:90,1] + 4.720;
   1:  PR[GP1:91,2] = PR[GP1:90,2] + 3.053;
   1:L PR[91] R[100]mm/sec CNT100;
   1:  PR[GP1:91,1] = PR[GP1:90,1] + 4.379;
   1:  PR[GP1:91,2] = PR[GP1:90,2] + 2.168;
   1:L PR[91] R[100]mm/sec CNT100;
   1:  PR[GP1:91,1] = PR[GP1:90,1] + 3.666;
   1:  PR[GP1:91,2] = PR[GP1:90,2] + 1.333;
   1:L PR[91] R[100]mm/sec CNT100;
   1:  PR[GP1:91,1] = PR[GP1:90,1] + 2.709;
   1:  PR[GP1:91,2] = PR[GP1:90,2] + 0.788;
   1:L PR[91] R[100]mm/sec CNT100;
   1:  PR[GP1:91,1] = PR[GP1:90,1] + 2.126;
   1:  PR[GP1:91,2] = PR[GP1:90,2] + 0.686;
   1:L PR[91] R[100]mm/sec CNT100;
   1:  PR[GP1:91,1] = PR[GP1:90,1] + 1.898;
   1:  PR[GP1:91,2] = PR[GP1:90,2] + 0.595;
   1:L PR[91] R[100]mm/sec CNT100;
   1:  PR[GP1:91,1] = PR[GP1:90,1] + -1.754;
   1:  PR[GP1:91,2] = PR[GP1:90,2] + 0.592;
   1:L PR[91] R[100]mm/sec CNT100;
   1:  PR[91] = PR[90];
   1:  PR[GP1:91,1] = PR[GP1:90,1] + -2.173;
   1:  PR[GP1:91,2] = PR[GP1:90,2] + 0.818;
   1:  PR[GP1:91,3] = PR[GP1:90,3] + 4.575;
   1:L PR[91] R[100]mm/sec CNT100;
   1:  PR[GP1:91,1] = PR[GP1:90,1] + -2.563;
   1:  PR[GP1:91,2] = PR[GP1:90,2] + 0.886;
   1:L PR[91] R[100]mm/sec CNT100;
   1:  PR[GP1:91,1] = PR[GP1:90,1] + -3.519;
   1:  PR[GP1:91,2] = PR[GP1:90,2] + 1.426;
   1:L PR[91] R[100]mm/sec CNT100;
   1:  PR[GP1:91,1] = PR[GP1:90,1] + -4.234;
   1:  PR[GP1:91,2] = PR[GP1:90,2] + 2.257;
   1:L PR[91] R[100]mm/sec CNT100;
   1:  PR[GP1:91,1] = PR[GP1:90,1] + -4.543;
   1:  PR[GP1:91,2] = PR[GP1:90,2] + 3.046;
   1:L PR[91] R[100]mm/sec CNT100;
   1:  PR[GP1:91,1] = PR[GP1:90,1] + -4.759;
   1:  PR[GP1:91,2] = PR[GP1:90,2] + 3.675;
   1:L PR[91] R[100]mm/sec CNT100;
